C09138=1210.781,-60.471,-39.584,179.733,5.457,149.035
C09139=1210.776,-60.222,-39.597,179.735,5.458,149.035
C09140=1210.771,-59.972,-39.609,179.737,5.458,149.034
C09141=1210.766,-59.722,-39.620,179.739,5.458,149.033
C09142=1210.761,-59.473,-39.632,179.742,5.459,149.033
C09143=1210.755,-59.223,-39.644,179.744,5.458,149.032
C09144=1210.751,-58.973,-39.655,179.747,5.459,149.031
C09145=1210.745,-58.724,-39.668,179.750,5.459,149.031
C09146=1210.740,-58.474,-39.679,179.752,5.459,149.030
C09147=1210.735,-58.224,-39.691,179.754,5.459,149.029
C09148=1210.730,-57.974,-39.703,179.756,5.459,149.029
C09149=1210.724,-57.724,-39.715,179.759,5.460,149.028
C09150=1210.720,-57.475,-39.726,179.761,5.460,149.027
C09151=1210.715,-57.225,-39.738,179.763,5.460,149.027
C09152=1210.709,-56.976,-39.750,179.766,5.460,149.026
C09153=1210.704,-56.726,-39.761,179.769,5.461,149.025
C09154=1210.699,-56.476,-39.773,179.771,5.460,149.025
C09155=1210.693,-56.227,-39.786,179.773,5.461,149.024
C09156=1210.689,-55.978,-39.797,179.776,5.460,149.023
C09157=1210.683,-55.728,-39.809,179.778,5.461,149.022
C09158=1210.678,-55.478,-39.821,179.780,5.462,149.022
C09159=1210.673,-55.229,-39.833,179.782,5.461,149.021
C09160=1210.668,-54.979,-39.845,179.785,5.462,149.021
C09161=1210.663,-54.729,-39.857,179.788,5.462,149.020
C09162=1210.657,-54.479,-39.868,179.790,5.462,149.019
C09163=1210.653,-54.230,-39.880,179.793,5.462,149.018
C09164=1210.647,-53.980,-39.892,179.795,5.462,149.018
C09165=1210.642,-53.730,-39.904,179.797,5.463,149.017
C09166=1210.637,-53.481,-39.917,179.800,5.463,149.016
C09167=1210.632,-53.231,-39.928,179.802,5.463,149.016
C09168=1210.627,-52.981,-39.940,179.804,5.464,149.015
C09169=1210.622,-52.732,-39.953,179.807,5.464,149.014
C09170=1210.616,-52.482,-39.964,179.809,5.464,149.014
C09171=1210.611,-52.232,-39.976,179.812,5.464,149.013
C09172=1210.606,-51.983,-39.988,179.814,5.464,149.012
C09173=1210.601,-51.733,-40.000,179.816,5.464,149.012
C09174=1210.596,-51.484,-40.013,179.819,5.465,149.011
C09175=1210.590,-51.234,-40.025,179.821,5.464,149.010
C09176=1210.586,-50.984,-40.036,179.824,5.465,149.010
C09177=1210.581,-50.735,-40.049,179.826,5.465,149.009
C09178=1210.575,-50.485,-40.060,179.828,5.465,149.008
C09179=1210.570,-50.236,-40.073,179.831,5.466,149.008
C09180=1210.565,-49.986,-40.085,179.833,5.466,149.007
C09181=1210.559,-49.736,-40.097,179.835,5.466,149.006
C09182=1210.555,-49.487,-40.109,179.838,5.466,149.006
C09183=1210.549,-49.216,-40.122,179.841,5.467,149.005
C09184=1210.543,-48.946,-40.135,179.843,5.466,149.004
C09185=1210.538,-48.677,-40.149,179.846,5.467,149.003
C09186=1210.532,-48.406,-40.162,179.849,5.467,149.002
C09187=1210.527,-48.156,-40.174,179.851,5.468,149.002
C09188=1210.522,-47.907,-40.186,179.853,5.467,149.001
C09189=1210.516,-47.657,-40.198,179.856,5.468,149.001
C09190=1210.511,-47.408,-40.211,179.858,5.468,149.000
C09191=1210.506,-47.158,-40.223,179.860,5.468,148.999
C09192=1210.502,-46.909,-40.235,179.863,5.469,148.998
C09193=1210.497,-46.658,-40.247,179.865,5.468,148.998
C09194=1210.492,-46.409,-40.259,179.868,5.469,148.997
C09195=1210.486,-46.159,-40.271,179.870,5.469,148.996
C09196=1210.481,-45.910,-40.284,179.873,5.469,148.996
C09197=1210.476,-45.660,-40.296,179.875,5.469,148.995
C09198=1210.470,-45.410,-40.308,179.877,5.470,148.995
C09199=1210.465,-45.161,-40.321,179.879,5.470,148.994
C09200=1210.460,-44.911,-40.333,179.882,5.470,148.993
C09201=1210.455,-44.662,-40.345,179.885,5.471,148.992
C09202=1210.449,-44.412,-40.357,179.887,5.470,148.992
C09203=1210.445,-44.162,-40.370,179.890,5.471,148.991
C09204=1210.440,-43.912,-40.383,179.892,5.471,148.990
C09205=1210.434,-43.663,-40.395,179.894,5.471,148.990
C09206=1210.429,-43.413,-40.407,179.897,5.471,148.989
C09207=1210.424,-43.163,-40.419,179.900,5.472,148.988
C09208=1210.419,-42.914,-40.432,179.901,5.472,148.988
C09209=1210.413,-42.665,-40.444,179.904,5.472,148.987
C09210=1210.409,-42.414,-40.457,179.907,5.473,148.986
C09211=1210.404,-42.165,-40.469,179.909,5.473,148.986
C09212=1210.398,-41.915,-40.482,179.911,5.473,148.985
C09213=1210.393,-41.665,-40.494,179.914,5.473,148.984
C09214=1210.388,-41.416,-40.506,179.916,5.473,148.984
C09215=1210.383,-41.167,-40.519,179.919,5.474,148.983
C09216=1210.378,-40.916,-40.531,179.921,5.474,148.982
C09217=1210.373,-40.667,-40.544,179.923,5.474,148.981
C09218=1210.368,-40.418,-40.556,179.926,5.474,148.981
C09219=1210.362,-40.168,-40.568,179.928,5.475,148.980
C09220=1210.357,-39.918,-40.581,179.930,5.475,148.980
C09221=1210.352,-39.669,-40.594,179.933,5.475,148.979
C09222=1210.347,-39.419,-40.607,179.936,5.476,148.978
C09223=1210.342,-39.169,-40.618,179.938,5.475,148.977
C09224=1210.337,-38.920,-40.631,179.940,5.476,148.977
C09225=1210.332,-38.670,-40.644,179.943,5.476,148.976
C09226=1210.327,-38.421,-40.656,179.945,5.476,148.975
C09227=1210.322,-38.170,-40.668,179.948,5.476,148.975
C09228=1210.317,-37.921,-40.681,179.950,5.477,148.974
C09229=1210.312,-37.672,-40.694,179.952,5.477,148.973
C09230=1210.306,-37.422,-40.707,179.955,5.477,148.973
C09231=1210.300,-37.172,-40.719,179.957,5.478,148.972
C09232=1210.296,-36.922,-40.732,179.959,5.477,148.971
C09233=1210.291,-36.673,-40.744,179.962,5.478,148.971
C09234=1210.286,-36.424,-40.757,179.965,5.478,148.970
C09235=1210.280,-36.174,-40.770,179.967,5.479,148.969
C09236=1210.276,-35.924,-40.782,179.970,5.479,148.969
C09237=1210.270,-35.674,-40.794,179.972,5.479,148.968
C09238=1210.265,-35.425,-40.808,179.975,5.480,148.967
C09239=1210.259,-35.175,-40.820,179.977,5.479,148.966
C09240=1210.255,-34.925,-40.833,179.979,5.480,148.966
C09241=1210.250,-34.676,-40.846,179.982,5.481,148.965
C09242=1210.245,-34.427,-40.858,179.984,5.480,148.965
C09243=1210.240,-34.177,-40.871,179.987,5.481,148.964
C09244=1210.234,-33.926,-40.884,179.989,5.481,148.963
C09245=1210.229,-33.677,-40.896,179.991,5.481,148.963
C09246=1210.224,-33.428,-40.909,179.994,5.481,148.962
C09247=1210.219,-33.178,-40.922,179.997,5.482,148.961
C09248=1210.214,-32.928,-40.935,179.999,5.482,148.960
C09249=1210.209,-32.679,-40.947,-179.999,5.482,148.960
C09250=1210.203,-32.430,-40.960,-179.996,5.482,148.959
C09251=1210.199,-32.179,-40.973,-179.994,5.483,148.959
C09252=1210.193,-31.930,-40.986,-179.992,5.483,148.958
C09253=1210.188,-31.681,-40.999,-179.989,5.483,148.957
C09254=1210.182,-31.431,-41.012,-179.986,5.484,148.956
C09255=1210.178,-31.181,-41.025,-179.984,5.484,148.956
C09256=1210.173,-30.932,-41.037,-179.982,5.484,148.955
C09257=1210.168,-30.683,-41.050,-179.979,5.484,148.954
C09258=1210.163,-30.433,-41.063,-179.976,5.485,148.954
C09259=1210.157,-30.183,-41.076,-179.974,5.485,148.953
C09260=1210.152,-29.934,-41.089,-179.972,5.485,148.952
C09261=1210.148,-29.684,-41.102,-179.969,5.486,148.952
C09262=1210.142,-29.434,-41.115,-179.967,5.486,148.951
C09263=1210.137,-29.185,-41.127,-179.965,5.486,148.950
C09264=1210.132,-28.935,-41.140,-179.962,5.487,148.950
C09265=1210.127,-28.685,-41.153,-179.960,5.486,148.949
C09266=1210.121,-28.436,-41.166,-179.957,5.487,148.948
C09267=1210.117,-28.186,-41.179,-179.955,5.487,148.948
C09268=1210.112,-27.936,-41.192,-179.952,5.488,148.947
C09269=1210.106,-27.687,-41.205,-179.950,5.487,148.946
C09270=1210.101,-27.437,-41.218,-179.947,5.488,148.946
C09271=1210.096,-27.187,-41.230,-179.945,5.488,148.945
C09272=1210.091,-26.939,-41.244,-179.942,5.489,148.944
C09273=1210.086,-26.688,-41.257,-179.940,5.489,148.944
C09274=1210.081,-26.439,-41.270,-179.938,5.489,148.943
C09275=1210.076,-26.189,-41.283,-179.935,5.490,148.942
C09276=1210.070,-25.939,-41.296,-179.933,5.489,148.942
C09277=1210.065,-25.690,-41.309,-179.930,5.490,148.941
C09278=1210.060,-25.440,-41.322,-179.928,5.490,148.940
C09279=1210.055,-25.190,-41.335,-179.925,5.491,148.939
C09280=1210.051,-24.941,-41.349,-179.923,5.491,148.939
C09281=1210.045,-24.691,-41.362,-179.920,5.491,148.938
C09282=1210.040,-24.442,-41.374,-179.918,5.492,148.937
C09283=1210.035,-24.192,-41.387,-179.916,5.492,148.937
C09284=1210.029,-23.942,-41.401,-179.913,5.492,148.936
C09285=1210.025,-23.693,-41.414,-179.911,5.493,148.936
C09286=1210.019,-23.443,-41.427,-179.908,5.493,148.935
C09287=1210.014,-23.174,-41.441,-179.905,5.494,148.934
C09288=1210.008,-22.905,-41.456,-179.903,5.493,148.933
C09289=1210.003,-22.635,-41.469,-179.900,5.493,148.933
C09290=1209.998,-22.365,-41.484,-179.897,5.494,148.932
C09291=1209.993,-22.117,-41.497,-179.895,5.494,148.931
C09292=1209.987,-21.866,-41.511,-179.892,5.495,148.930
C09293=1209.982,-21.617,-41.523,-179.891,5.495,148.930
C09294=1209.977,-21.367,-41.537,-179.888,5.495,148.929
C09295=1209.972,-21.118,-41.550,-179.885,5.496,148.929
C09296=1209.966,-20.868,-41.563,-179.883,5.496,148.928
C09297=1209.962,-20.618,-41.576,-179.880,5.496,148.927
C09298=1209.956,-20.369,-41.590,-179.878,5.496,148.926
C09299=1209.952,-20.119,-41.603,-179.875,5.497,148.926
C09300=1209.946,-19.870,-41.616,-179.872,5.497,148.925
C09301=1209.942,-19.620,-41.630,-179.870,5.497,148.924
C09302=1209.937,-19.371,-41.643,-179.868,5.498,148.924
C09303=1209.931,-19.120,-41.656,-179.865,5.498,148.923
C09304=1209.926,-18.872,-41.669,-179.863,5.499,148.923
C09305=1209.921,-18.621,-41.683,-179.861,5.499,148.922
C09306=1209.915,-18.372,-41.696,-179.858,5.499,148.921
C09307=1209.911,-18.122,-41.710,-179.856,5.500,148.920
C09308=1209.905,-17.873,-41.723,-179.853,5.500,148.920
C09309=1209.901,-17.623,-41.736,-179.851,5.500,148.919
C09310=1209.895,-17.374,-41.750,-179.848,5.500,148.918
C09311=1209.891,-17.124,-41.763,-179.845,5.501,148.918
C09312=1209.885,-16.875,-41.777,-179.843,5.501,148.917
C09313=1209.881,-16.625,-41.790,-179.841,5.501,148.916
C09314=1209.875,-16.376,-41.804,-179.839,5.502,148.916
C09315=1209.871,-16.126,-41.817,-179.836,5.502,148.915
C09316=1209.865,-15.876,-41.830,-179.833,5.503,148.914
C09317=1209.860,-15.627,-41.844,-179.831,5.502,148.914
C09318=1209.855,-15.377,-41.857,-179.829,5.503,148.913
C09319=1209.850,-15.127,-41.871,-179.826,5.503,148.912
C09320=1209.844,-14.878,-41.884,-179.823,5.504,148.912
C09321=1209.840,-14.628,-41.898,-179.821,5.504,148.911
C09322=1209.834,-14.379,-41.910,-179.818,5.504,148.910
C09323=1209.829,-14.129,-41.925,-179.816,5.505,148.910
C09324=1209.824,-13.879,-41.938,-179.814,5.505,148.909
C09325=1209.819,-13.630,-41.952,-179.811,5.506,148.908
C09326=1209.814,-13.380,-41.965,-179.809,5.506,148.908
C09327=1209.809,-13.131,-41.979,-179.806,5.506,148.907
C09328=1209.804,-12.881,-41.992,-179.804,5.507,148.906
C09329=1209.798,-12.632,-42.006,-179.801,5.507,148.906
C09330=1209.794,-12.382,-42.019,-179.799,5.507,148.905
C09331=1209.789,-12.132,-42.033,-179.796,5.507,148.904
C09332=1209.783,-11.883,-42.047,-179.794,5.508,148.904
C09333=1209.779,-11.633,-42.060,-179.791,5.508,148.903
C09334=1209.773,-11.384,-42.074,-179.789,5.508,148.902
C09335=1209.768,-11.134,-42.088,-179.787,5.509,148.902
C09336=1209.763,-10.885,-42.101,-179.784,5.509,148.901
C09337=1209.758,-10.635,-42.115,-179.781,5.510,148.900
C09338=1209.753,-10.385,-42.129,-179.779,5.510,148.900
C09339=1209.748,-10.136,-42.142,-179.777,5.510,148.899
C09340=1209.743,-9.886,-42.156,-179.774,5.510,148.898
C09341=1209.738,-9.636,-42.170,-179.771,5.511,148.898
C09342=1209.733,-9.388,-42.183,-179.769,5.511,148.897
C09343=1209.728,-9.137,-42.197,-179.766,5.512,148.896
C09344=1209.722,-8.888,-42.211,-179.764,5.512,148.896
C09345=1209.717,-8.639,-42.225,-179.762,5.512,148.895
C09346=1209.713,-8.389,-42.238,-179.759,5.513,148.894
C09347=1209.707,-8.140,-42.252,-179.756,5.513,148.894
C09348=1209.702,-7.890,-42.266,-179.754,5.513,148.893
C09349=1209.697,-7.639,-42.280,-179.752,5.514,148.892
C09350=1209.692,-7.391,-42.293,-179.749,5.514,148.892
C09351=1209.687,-7.141,-42.307,-179.746,5.515,148.891
C09352=1209.682,-6.891,-42.322,-179.744,5.515,148.890
C09353=1209.677,-6.642,-42.335,-179.742,5.515,148.890
C09354=1209.672,-6.392,-42.348,-179.739,5.516,148.889
C09355=1209.667,-6.143,-42.363,-179.737,5.516,148.888
C09356=1209.662,-5.894,-42.377,-179.734,5.517,148.888
C09357=1209.657,-5.643,-42.390,-179.732,5.517,148.887
C09358=1209.652,-5.394,-42.404,-179.729,5.517,148.886
C09359=1209.647,-5.145,-42.418,-179.727,5.517,148.886
C09360=1209.642,-4.895,-42.432,-179.724,5.518,148.885
C09361=1209.637,-4.645,-42.446,-179.721,5.518,148.884
C09362=1209.631,-4.396,-42.460,-179.719,5.519,148.884
C09363=1209.626,-4.146,-42.474,-179.717,5.520,148.883
C09364=1209.622,-3.897,-42.487,-179.715,5.519,148.882
C09365=1209.616,-3.648,-42.501,-179.712,5.520,148.882
C09366=1209.611,-3.397,-42.515,-179.709,5.520,148.881
C09367=1209.606,-3.148,-42.529,-179.707,5.521,148.880
C09368=1209.601,-2.898,-42.544,-179.704,5.521,148.880
C09369=1209.596,-2.649,-42.557,-179.702,5.521,148.879
C09370=1209.591,-2.400,-42.571,-179.699,5.522,148.878
C09371=1209.586,-2.150,-42.585,-179.697,5.522,148.878
C09372=1209.581,-1.901,-42.599,-179.694,5.523,148.877
C09373=1209.576,-1.651,-42.614,-179.692,5.523,148.876
C09374=1209.571,-1.401,-42.627,-179.690,5.523,148.876
C09375=1209.566,-1.151,-42.641,-179.687,5.524,148.875
C09376=1209.560,-0.902,-42.655,-179.684,5.524,148.874
C09377=1209.555,-0.652,-42.670,-179.682,5.525,148.874
C09378=1209.550,-0.403,-42.684,-179.679,5.525,148.873
C09379=1209.546,-0.153,-42.698,-179.676,5.526,148.872
C09380=1209.540,0.096,-42.711,-179.674,5.525,148.872
C09381=1209.536,0.345,-42.726,-179.672,5.526,148.871
C09382=1209.531,0.595,-42.740,-179.670,5.527,148.870
C09383=1209.526,0.845,-42.754,-179.667,5.527,148.870
C09384=1209.520,1.094,-42.768,-179.664,5.528,148.869
C09385=1209.515,1.344,-42.782,-179.662,5.528,148.868
C09386=1209.510,1.593,-42.797,-179.660,5.528,148.868
C09387=1209.505,1.843,-42.811,-179.657,5.528,148.867
C09388=1209.500,2.093,-42.825,-179.654,5.529,148.866
C09389=1209.495,2.342,-42.839,-179.652,5.529,148.866
C09390=1209.490,2.591,-42.854,-179.649,5.530,148.865
C09391=1209.484,2.861,-42.869,-179.646,5.530,148.864
C09392=1209.479,3.130,-42.884,-179.644,5.531,148.864
C09393=1209.474,3.399,-42.899,-179.641,5.532,148.863
C09394=1209.469,3.668,-42.915,-179.638,5.532,148.862
C09395=1209.463,3.917,-42.929,-179.636,5.532,148.861
C09396=1209.458,4.167,-42.943,-179.634,5.532,148.861
C09397=1209.453,4.416,-42.957,-179.631,5.533,148.860
C09398=1209.448,4.666,-42.972,-179.629,5.534,148.860
C09399=1209.443,4.916,-42.986,-179.626,5.534,148.859
C09400=1209.438,5.165,-43.000,-179.623,5.535,148.858
C09401=1209.433,5.414,-43.014,-179.621,5.535,148.858
C09402=1209.428,5.664,-43.029,-179.619,5.535,148.857
C09403=1209.423,5.913,-43.043,-179.616,5.535,148.856
C09404=1209.417,6.163,-43.058,-179.613,5.536,148.856
C09405=1209.412,6.413,-43.073,-179.611,5.536,148.855
C09406=1209.407,6.663,-43.087,-179.609,5.537,148.854
C09407=1209.403,6.912,-43.101,-179.606,5.538,148.854
C09408=1209.397,7.161,-43.115,-179.603,5.538,148.853
C09409=1209.392,7.411,-43.130,-179.601,5.538,148.852
C09410=1209.387,7.660,-43.144,-179.599,5.538,148.852
C09411=1209.382,7.910,-43.159,-179.596,5.539,148.851
C09412=1209.377,8.160,-43.173,-179.593,5.539,148.850
C09413=1209.373,8.409,-43.187,-179.591,5.540,148.850
C09414=1209.368,8.658,-43.202,-179.588,5.541,148.849
C09415=1209.363,8.908,-43.216,-179.586,5.541,148.848
C09416=1209.357,9.157,-43.231,-179.584,5.541,148.848
C09417=1209.352,9.407,-43.245,-179.581,5.542,148.847
C09418=1209.347,9.656,-43.260,-179.578,5.542,148.846
C09419=1209.342,9.906,-43.274,-179.576,5.543,148.846
C09420=1209.337,10.156,-43.289,-179.573,5.543,148.845
C09421=1209.332,10.405,-43.303,-179.571,5.544,148.845
C09422=1209.328,10.654,-43.318,-179.568,5.544,148.844
C09423=1209.322,10.905,-43.333,-179.566,5.544,148.843
C09424=1209.317,11.154,-43.347,-179.564,5.545,148.843
C09425=1209.312,11.403,-43.362,-179.561,5.545,148.842
C09426=1209.307,11.653,-43.376,-179.558,5.546,148.841
C09427=1209.302,11.902,-43.390,-179.556,5.546,148.840
C09428=1209.296,12.152,-43.405,-179.553,5.547,148.840
C09429=1209.291,12.401,-43.420,-179.551,5.548,148.839
C09430=1209.286,12.651,-43.434,-179.548,5.548,148.839
C09431=1209.282,12.900,-43.449,-179.546,5.549,148.838
C09432=1209.277,13.150,-43.464,-179.543,5.548,148.837
C09433=1209.271,13.400,-43.479,-179.541,5.549,148.837
C09434=1209.266,13.649,-43.494,-179.538,5.549,148.836
C09435=1209.262,13.898,-43.508,-179.536,5.550,148.835
C09436=1209.257,14.148,-43.522,-179.533,5.551,148.835
C09437=1209.252,14.397,-43.537,-179.531,5.551,148.834
C09438=1209.246,14.647,-43.552,-179.528,5.552,148.833
C09439=1209.242,14.896,-43.567,-179.525,5.552,148.833
C09440=1209.237,15.146,-43.581,-179.523,5.552,148.832
C09441=1209.231,15.396,-43.597,-179.521,5.553,148.831
C09442=1209.226,15.645,-43.611,-179.518,5.553,148.831
C09443=1209.221,15.895,-43.625,-179.516,5.554,148.830
C09444=1209.217,16.144,-43.640,-179.513,5.554,148.830
C09445=1209.211,16.394,-43.655,-179.511,5.555,148.829
C09446=1209.206,16.643,-43.670,-179.508,5.556,148.828
C09447=1209.201,16.893,-43.685,-179.505,5.556,148.827
C09448=1209.196,17.142,-43.700,-179.503,5.557,148.827
C09449=1209.191,17.392,-43.714,-179.500,5.557,148.826
C09450=1209.186,17.641,-43.729,-179.498,5.557,148.825
C09451=1209.181,17.891,-43.744,-179.496,5.558,148.825
C09452=1209.176,18.140,-43.759,-179.493,5.558,148.824
C09453=1209.171,18.390,-43.774,-179.490,5.559,148.824
C09454=1209.166,18.639,-43.789,-179.488,5.559,148.823
C09455=1209.161,18.889,-43.803,-179.485,5.560,148.822
C09456=1209.156,19.138,-43.818,-179.483,5.560,148.822
C09457=1209.151,19.387,-43.834,-179.480,5.561,148.821
C09458=1209.146,19.637,-43.848,-179.478,5.562,148.820
C09459=1209.141,19.886,-43.863,-179.475,5.562,148.820
C09460=1209.135,20.136,-43.878,-179.472,5.563,148.819
C09461=1209.131,20.385,-43.893,-179.470,5.562,148.818
C09462=1209.127,20.635,-43.908,-179.468,5.563,148.818
C09463=1209.121,20.885,-43.923,-179.465,5.563,148.817
C09464=1209.116,21.134,-43.938,-179.463,5.564,148.817
C09465=1209.111,21.384,-43.953,-179.460,5.565,148.816
C09466=1209.106,21.633,-43.968,-179.458,5.565,148.815
C09467=1209.101,21.883,-43.983,-179.455,5.566,148.815
C09468=1209.096,22.133,-43.998,-179.452,5.566,148.814
C09469=1209.091,22.382,-44.013,-179.450,5.567,148.813
C09470=1209.086,22.631,-44.029,-179.447,5.567,148.812
C09471=1209.081,22.881,-44.043,-179.445,5.568,148.812
C09472=1209.075,23.130,-44.059,-179.442,5.569,148.811
C09473=1209.071,23.380,-44.074,-179.440,5.569,148.811
C09474=1209.066,23.630,-44.088,-179.438,5.569,148.810
C09475=1209.061,23.879,-44.104,-179.435,5.570,148.809
C09476=1209.056,24.128,-44.119,-179.432,5.570,148.809
C09477=1209.051,24.378,-44.134,-179.430,5.571,148.808
C09478=1209.046,24.627,-44.149,-179.427,5.572,148.807
C09479=1209.041,24.877,-44.164,-179.425,5.572,148.807
C09480=1209.036,25.126,-44.179,-179.422,5.573,148.806
C09481=1209.031,25.376,-44.195,-179.419,5.573,148.805
C09482=1209.026,25.626,-44.209,-179.417,5.574,148.805
C09483=1209.021,25.875,-44.225,-179.415,5.575,148.804
C09484=1209.016,26.124,-44.240,-179.412,5.575,148.804
C09485=1209.011,26.373,-44.256,-179.409,5.576,148.803
C09486=1209.006,26.623,-44.271,-179.407,5.576,148.802
C09487=1209.000,26.873,-44.285,-179.404,5.577,148.802
C09488=1208.996,27.122,-44.301,-179.401,5.577,148.801
C09489=1208.991,27.372,-44.316,-179.399,5.578,148.800
C09490=1208.986,27.621,-44.332,-179.397,5.578,148.800
C09491=1208.981,27.870,-44.347,-179.395,5.578,148.799
C09492=1208.976,28.120,-44.363,-179.392,5.579,148.798
C09493=1208.971,28.369,-44.377,-179.389,5.579,148.798
C09494=1208.966,28.619,-44.393,-179.387,5.580,148.797
C09495=1208.961,28.888,-44.409,-179.384,5.580,148.796
C09496=1208.955,29.157,-44.426,-179.381,5.582,148.796
C09497=1208.950,29.425,-44.443,-179.378,5.582,148.795
C09498=1208.944,29.694,-44.458,-179.375,5.583,148.794
C09499=1208.939,29.943,-44.474,-179.373,5.583,148.794
C09500=1208.934,30.193,-44.489,-179.371,5.584,148.793
C09501=1208.930,30.443,-44.505,-179.368,5.585,148.793
C09502=1208.924,30.692,-44.520,-179.365,5.585,148.792
C09503=1208.920,30.941,-44.535,-179.363,5.586,148.791
C09504=1208.914,31.191,-44.551,-179.361,5.586,148.791
C09505=1208.909,31.440,-44.567,-179.358,5.586,148.790
C09506=1208.905,31.690,-44.582,-179.356,5.587,148.789
C09507=1208.899,31.939,-44.597,-179.353,5.587,148.789
C09508=1208.894,32.189,-44.613,-179.351,5.588,148.788
C09509=1208.889,32.438,-44.628,-179.348,5.589,148.787
C09510=1208.885,32.688,-44.644,-179.345,5.589,148.787
C09511=1208.879,32.937,-44.660,-179.343,5.590,148.786
C09512=1208.874,33.186,-44.675,-179.341,5.590,148.786
C09513=1208.869,33.436,-44.690,-179.338,5.591,148.785
C09514=1208.864,33.686,-44.706,-179.335,5.592,148.784
C09515=1208.860,33.935,-44.721,-179.333,5.592,148.784
C09516=1208.854,34.184,-44.737,-179.330,5.593,148.783
C09517=1208.849,34.434,-44.753,-179.328,5.594,148.782
C09518=1208.845,34.683,-44.768,-179.325,5.594,148.782
C09519=1208.839,34.933,-44.783,-179.323,5.595,148.781
C09520=1208.834,35.182,-44.800,-179.320,5.595,148.780
C09521=1208.830,35.432,-44.816,-179.317,5.596,148.780
C09522=1208.825,35.681,-44.831,-179.315,5.597,148.779
C09523=1208.820,35.930,-44.846,-179.312,5.597,148.779
C09524=1208.815,36.180,-44.862,-179.310,5.598,148.778
C09525=1208.809,36.430,-44.878,-179.307,5.598,148.777
C09526=1208.805,36.679,-44.893,-179.305,5.599,148.777
C09527=1208.800,36.929,-44.909,-179.302,5.600,148.776
C09528=1208.795,37.178,-44.925,-179.300,5.600,148.775
C09529=1208.789,37.427,-44.940,-179.297,5.601,148.775
C09530=1208.784,37.676,-44.956,-179.294,5.601,148.774
C09531=1208.780,37.926,-44.971,-179.292,5.602,148.773
C09532=1208.775,38.176,-44.987,-179.289,5.602,148.773
C09533=1208.769,38.425,-45.003,-179.287,5.603,148.772
C09534=1208.765,38.675,-45.019,-179.284,5.604,148.772
C09535=1208.759,38.924,-45.035,-179.282,5.604,148.771
C09536=1208.755,39.173,-45.050,-179.279,5.605,148.770
C09537=1208.750,39.423,-45.066,-179.276,5.605,148.770
C09538=1208.745,39.672,-45.082,-179.274,5.606,148.769
C09539=1208.740,39.922,-45.098,-179.272,5.607,148.769
C09540=1208.735,40.171,-45.114,-179.269,5.607,148.768
C09541=1208.729,40.421,-45.129,-179.266,5.608,148.767
C09542=1208.726,40.670,-45.145,-179.264,5.608,148.766
C09543=1208.720,40.919,-45.161,-179.262,5.609,148.766
C09544=1208.715,41.169,-45.176,-179.259,5.610,148.765
C09545=1208.710,41.419,-45.192,-179.256,5.610,148.765
C09546=1208.705,41.668,-45.209,-179.254,5.611,148.764
C09547=1208.700,41.918,-45.225,-179.251,5.611,148.763
C09548=1208.695,42.167,-45.240,-179.249,5.612,148.763
C09549=1208.690,42.416,-45.257,-179.246,5.613,148.762
C09550=1208.685,42.666,-45.273,-179.244,5.613,148.762
C09551=1208.680,42.915,-45.288,-179.241,5.614,148.761
C09552=1208.676,43.165,-45.304,-179.239,5.615,148.760
C09553=1208.670,43.414,-45.320,-179.236,5.615,148.760
C09554=1208.665,43.663,-45.336,-179.234,5.616,148.759
C09555=1208.661,43.913,-45.352,-179.231,5.616,148.758
C09556=1208.655,44.162,-45.368,-179.228,5.617,148.758
C09557=1208.651,44.412,-45.384,-179.226,5.618,148.757
C09558=1208.645,44.661,-45.400,-179.223,5.618,148.757
C09559=1208.641,44.911,-45.417,-179.221,5.619,148.756
C09560=1208.635,45.160,-45.432,-179.218,5.619,148.755
C09561=1208.630,45.410,-45.448,-179.215,5.621,148.755
C09562=1208.626,45.659,-45.464,-179.213,5.622,148.754
C09563=1208.620,45.908,-45.480,-179.210,5.622,148.754
C09564=1208.616,46.158,-45.497,-179.208,5.623,148.753
C09565=1208.610,46.407,-45.512,-179.205,5.623,148.752
C09566=1208.606,46.657,-45.529,-179.203,5.624,148.752
C09567=1208.600,46.906,-45.545,-179.200,5.625,148.751
C09568=1208.596,47.156,-45.561,-179.197,5.625,148.750
C09569=1208.591,47.405,-45.577,-179.195,5.626,148.750
C09570=1208.586,47.655,-45.593,-179.192,5.626,148.749
C09571=1208.581,47.904,-45.609,-179.190,5.627,148.749
C09572=1208.576,48.153,-45.626,-179.187,5.628,148.748
C09573=1208.571,48.403,-45.641,-179.185,5.628,148.747
C09574=1208.566,48.652,-45.658,-179.182,5.629,148.747
C09575=1208.561,48.902,-45.674,-179.180,5.630,148.746
C09576=1208.556,49.151,-45.690,-179.177,5.630,148.745
C09577=1208.551,49.400,-45.707,-179.175,5.631,148.745
C09578=1208.547,49.650,-45.722,-179.172,5.631,148.744
C09579=1208.542,49.899,-45.739,-179.170,5.632,148.744
C09580=1208.537,50.149,-45.755,-179.167,5.633,148.743
C09581=1208.532,50.398,-45.771,-179.165,5.633,148.742
C09582=1208.527,50.647,-45.788,-179.161,5.635,148.742
C09583=1208.521,50.897,-45.804,-179.159,5.635,148.741
C09584=1208.517,51.146,-45.821,-179.157,5.636,148.741
C09585=1208.511,51.396,-45.836,-179.154,5.637,148.740
C09586=1208.507,51.645,-45.853,-179.151,5.637,148.739
C09587=1208.502,51.894,-45.869,-179.149,5.638,148.739
C09588=1208.497,52.144,-45.885,-179.147,5.639,148.738
C09589=1208.492,52.394,-45.902,-179.144,5.639,148.737
C09590=1208.487,52.642,-45.918,-179.141,5.640,148.737
C09591=1208.482,52.893,-45.935,-179.139,5.640,148.736
C09592=1208.477,53.142,-45.951,-179.137,5.641,148.736
C09593=1208.472,53.391,-45.968,-179.134,5.642,148.735
C09594=1208.467,53.640,-45.984,-179.131,5.642,148.734
C09595=1208.462,53.890,-46.000,-179.129,5.643,148.734
C09596=1208.458,54.140,-46.016,-179.126,5.645,148.733
C09597=1208.452,54.389,-46.033,-179.123,5.645,148.733
C09598=1208.448,54.638,-46.050,-179.121,5.646,148.732
C09599=1208.442,54.907,-46.067,-179.118,5.646,148.731
C09600=1208.437,55.175,-46.085,-179.115,5.647,148.731
C09601=1208.431,55.444,-46.103,-179.113,5.648,148.730
C09602=1208.426,55.712,-46.121,-179.110,5.649,148.729
C09603=1208.421,55.961,-46.137,-179.107,5.650,148.729
C09604=1208.417,56.211,-46.154,-179.105,5.650,148.728
C09605=1208.411,56.460,-46.170,-179.102,5.651,148.727
C09606=1208.406,56.710,-46.187,-179.099,5.651,148.727
C09607=1208.401,56.959,-46.203,-179.097,5.652,148.726
C09608=1208.397,57.208,-46.220,-179.095,5.653,148.726
C09609=1208.391,57.458,-46.237,-179.092,5.653,148.725
C09610=1208.386,57.707,-46.253,-179.089,5.654,148.724
C09611=1208.382,57.957,-46.269,-179.087,5.656,148.724
C09612=1208.377,58.206,-46.286,-179.084,5.656,148.723
C09613=1208.371,58.456,-46.303,-179.081,5.657,148.723
C09614=1208.367,58.705,-46.319,-179.079,5.657,148.722
C09615=1208.362,58.954,-46.336,-179.077,5.658,148.722
C09616=1208.357,59.204,-46.353,-179.074,5.659,148.721
C09617=1208.352,59.453,-46.370,-179.071,5.659,148.720
C09618=1208.348,59.703,-46.386,-179.069,5.660,148.720
C09619=1208.342,59.951,-46.403,-179.067,5.661,148.719
C09620=1208.337,60.201,-46.420,-179.064,5.661,148.718
C09621=1208.333,60.451,-46.437,-179.061,5.663,148.718
C09622=1208.328,60.699,-46.453,-179.059,5.664,148.717
C09623=1208.322,60.949,-46.470,-179.056,5.664,148.717
C09624=1208.318,61.199,-46.487,-179.053,5.665,148.716
C09625=1208.312,61.448,-46.504,-179.051,5.665,148.715
C09626=1208.308,61.697,-46.520,-179.049,5.666,148.715
C09627=1208.303,61.947,-46.537,-179.046,5.667,148.714
C09628=1208.298,62.197,-46.554,-179.043,5.667,148.714
C09629=1208.293,62.445,-46.571,-179.040,5.669,148.713
C09630=1208.288,62.695,-46.587,-179.038,5.670,148.712
C09631=1208.283,62.945,-46.605,-179.035,5.670,148.712
C09632=1208.278,63.193,-46.621,-179.033,5.671,148.711
C09633=1208.273,63.443,-46.638,-179.031,5.672,148.711
C09634=1208.268,63.693,-46.655,-179.028,5.672,148.710
C09635=1208.264,63.942,-46.671,-179.025,5.673,148.709
C09636=1208.258,64.191,-46.688,-179.023,5.673,148.709
C09637=1208.254,64.441,-46.705,-179.020,5.675,148.708
C09638=1208.248,64.691,-46.722,-179.017,5.676,148.708
C09639=1208.244,64.940,-46.739,-179.015,5.676,148.707
C09640=1208.238,65.189,-46.756,-179.013,5.677,148.707
C09641=1208.234,65.438,-46.773,-179.010,5.678,148.706
C09642=1208.229,65.687,-46.790,-179.007,5.678,148.705
C09643=1208.224,65.937,-46.807,-179.005,5.679,148.705
C09644=1208.219,66.186,-46.823,-179.002,5.681,148.704
C09645=1208.214,66.436,-46.841,-178.999,5.681,148.703
C09646=1208.209,66.685,-46.857,-178.997,5.682,148.703
C09647=1208.205,66.934,-46.875,-178.995,5.683,148.702
C09648=1208.200,67.184,-46.892,-178.992,5.683,148.702
C09649=1208.194,67.433,-46.909,-178.989,5.684,148.701
C09650=1208.190,67.683,-46.926,-178.987,5.684,148.700
C09651=1208.185,67.932,-46.943,-178.984,5.686,148.700
C09652=1208.180,68.181,-46.960,-178.981,5.687,148.699
C09653=1208.175,68.431,-46.978,-178.979,5.687,148.699
C09654=1208.170,68.680,-46.994,-178.977,5.688,148.698
C09655=1208.165,68.930,-47.011,-178.974,5.689,148.698
C09656=1208.161,69.178,-47.028,-178.971,5.689,148.697
C09657=1208.155,69.428,-47.046,-178.969,5.691,148.696
C09658=1208.150,69.678,-47.063,-178.966,5.691,148.696
C09659=1208.146,69.927,-47.080,-178.963,5.692,148.695
C09660=1208.140,70.176,-47.097,-178.961,5.693,148.694
C09661=1208.136,70.425,-47.114,-178.959,5.693,148.694
C09662=1208.131,70.675,-47.131,-178.956,5.694,148.693
C09663=1208.126,70.924,-47.149,-178.953,5.695,148.693
C09664=1208.121,71.174,-47.166,-178.951,5.696,148.692
C09665=1208.116,71.424,-47.183,-178.948,5.697,148.692
C09666=1208.112,71.673,-47.201,-178.945,5.697,148.691
C09667=1208.106,71.922,-47.217,-178.943,5.698,148.691
C09668=1208.101,72.171,-47.235,-178.941,5.699,148.690
C09669=1208.097,72.420,-47.252,-178.937,5.700,148.689
C09670=1208.091,72.670,-47.269,-178.935,5.701,148.689
C09671=1208.087,72.919,-47.287,-178.933,5.702,148.688
C09672=1208.082,73.169,-47.304,-178.930,5.702,148.687
C09673=1208.077,73.418,-47.322,-178.928,5.703,148.687
C09674=1208.073,73.667,-47.339,-178.925,5.704,148.686
C09675=1208.067,73.917,-47.356,-178.922,5.705,148.686
C09676=1208.062,74.166,-47.374,-178.920,5.706,148.685
C09677=1208.057,74.415,-47.390,-178.917,5.707,148.685
C09678=1208.052,74.664,-47.408,-178.915,5.707,148.684
C09679=1208.047,74.914,-47.425,-178.912,5.708,148.684
C09680=1208.043,75.163,-47.443,-178.909,5.710,148.683
C09681=1208.038,75.413,-47.460,-178.907,5.710,148.682
C09682=1208.033,75.662,-47.478,-178.904,5.711,148.682
C09683=1208.028,75.912,-47.495,-178.902,5.712,148.681
C09684=1208.024,76.161,-47.513,-178.899,5.712,148.681
C09685=1208.018,76.410,-47.530,-178.896,5.714,148.680
C09686=1208.013,76.660,-47.548,-178.894,5.715,148.679
C09687=1208.009,76.909,-47.565,-178.891,5.715,148.679
C09688=1208.004,77.158,-47.583,-178.889,5.716,148.678
C09689=1207.999,77.408,-47.600,-178.886,5.717,148.678
C09690=1207.994,77.657,-47.618,-178.883,5.718,148.677
C09691=1207.989,77.905,-47.635,-178.881,5.719,148.677
C09692=1207.984,78.155,-47.652,-178.879,5.719,148.676
C09693=1207.979,78.404,-47.670,-178.876,5.720,148.675
C09694=1207.974,78.654,-47.687,-178.874,5.721,148.675
C09695=1207.969,78.903,-47.705,-178.871,5.722,148.674
C09696=1207.965,79.152,-47.723,-178.868,5.723,148.674
C09697=1207.959,79.402,-47.740,-178.866,5.724,148.673
C09698=1207.955,79.651,-47.758,-178.863,5.724,148.672
C09699=1207.950,79.900,-47.776,-178.861,5.725,148.672
C09700=1207.944,80.150,-47.793,-178.858,5.727,148.671
C09701=1207.940,80.399,-47.811,-178.855,5.727,148.671
C09702=1207.935,80.648,-47.829,-178.853,5.728,148.670
C09703=1207.930,80.917,-47.847,-178.849,5.729,148.669
C09704=1207.925,81.185,-47.867,-178.847,5.730,148.669
C09705=1207.919,81.454,-47.885,-178.845,5.731,148.668
C09706=1207.914,81.722,-47.905,-178.841,5.732,148.668
C09707=1207.909,81.972,-47.923,-178.839,5.733,148.667
C09708=1207.904,82.221,-47.940,-178.837,5.734,148.667
C09709=1207.899,82.471,-47.958,-178.834,5.734,148.666
C09710=1207.894,82.720,-47.976,-178.831,5.736,148.665
C09711=1207.890,82.969,-47.993,-178.829,5.737,148.665
C09712=1207.885,83.218,-48.011,-178.826,5.737,148.664
C09713=1207.880,83.468,-48.029,-178.823,5.738,148.664
C09714=1207.875,83.717,-48.047,-178.821,5.739,148.663
C09715=1207.870,83.966,-48.065,-178.818,5.740,148.663
C09716=1207.865,84.215,-48.083,-178.816,5.741,148.662
C09717=1207.860,84.465,-48.100,-178.813,5.741,148.661
C09718=1207.855,84.714,-48.118,-178.810,5.743,148.661
C09719=1207.850,84.963,-48.136,-178.808,5.744,148.660
C09720=1207.846,85.213,-48.154,-178.805,5.744,148.660
C09721=1207.841,85.462,-48.172,-178.803,5.745,148.659
C09722=1207.836,85.712,-48.190,-178.800,5.747,148.659
C09723=1207.831,85.961,-48.208,-178.797,5.747,148.658
C09724=1207.826,86.210,-48.225,-178.795,5.748,148.658
C09725=1207.821,86.460,-48.243,-178.793,5.749,148.657
C09726=1207.816,86.709,-48.261,-178.789,5.750,148.656
C09727=1207.811,86.958,-48.279,-178.787,5.751,148.656
C09728=1207.806,87.207,-48.297,-178.785,5.752,148.655
C09729=1207.802,87.456,-48.315,-178.782,5.752,148.655
C09730=1207.797,87.706,-48.334,-178.779,5.754,148.654
C09731=1207.792,87.955,-48.352,-178.777,5.755,148.653
C09732=1207.787,88.205,-48.370,-178.775,5.755,148.653
C09733=1207.782,88.454,-48.388,-178.772,5.756,148.652
C09734=1207.778,88.703,-48.406,-178.769,5.757,148.652
C09735=1207.773,88.952,-48.423,-178.767,5.758,148.651
C09736=1207.768,89.201,-48.441,-178.764,5.759,148.651
C09737=1207.763,89.451,-48.460,-178.761,5.761,148.650
C09738=1207.759,89.700,-48.478,-178.759,5.761,148.650
C09739=1207.754,89.950,-48.496,-178.756,5.762,148.649
C09740=1207.749,90.199,-48.514,-178.754,5.763,148.649
C09741=1207.744,90.448,-48.532,-178.751,5.764,148.648
C09742=1207.739,90.697,-48.550,-178.749,5.765,148.647
C09743=1207.735,90.947,-48.568,-178.746,5.766,148.647
C09744=1207.730,91.196,-48.586,-178.743,5.766,148.646
C09745=1207.724,91.446,-48.605,-178.741,5.768,148.646
C09746=1207.719,91.695,-48.623,-178.738,5.769,148.645
C09747=1207.714,91.944,-48.641,-178.736,5.770,148.645
C09748=1207.709,92.193,-48.659,-178.733,5.771,148.644
C09749=1207.705,92.443,-48.677,-178.730,5.772,148.643
C09750=1207.700,92.692,-48.696,-178.728,5.772,148.643
C09751=1207.695,92.941,-48.714,-178.725,5.773,148.642
C09752=1207.691,93.190,-48.732,-178.723,5.775,148.642
C09753=1207.685,93.440,-48.751,-178.720,5.775,148.641
C09754=1207.681,93.689,-48.768,-178.717,5.776,148.641
C09755=1207.676,93.938,-48.786,-178.715,5.778,148.640
C09756=1207.671,94.188,-48.804,-178.712,5.778,148.640
C09757=1207.666,94.436,-48.823,-178.710,5.779,148.639
C09758=1207.662,94.686,-48.841,-178.707,5.781,148.638
C09759=1207.656,94.936,-48.860,-178.704,5.781,148.638
C09760=1207.651,95.185,-48.878,-178.702,5.782,148.637
C09761=1207.646,95.434,-48.896,-178.699,5.783,148.637
C09762=1207.642,95.683,-48.915,-178.697,5.784,148.636
C09763=1207.637,95.933,-48.934,-178.694,5.785,148.636
C09764=1207.632,96.182,-48.952,-178.692,5.786,148.635
C09765=1207.627,96.431,-48.970,-178.689,5.787,148.635
C09766=1207.623,96.680,-48.989,-178.686,5.788,148.634
C09767=1207.618,96.929,-49.007,-178.684,5.789,148.634
C09768=1207.612,97.179,-49.025,-178.681,5.790,148.633
C09769=1207.608,97.428,-49.044,-178.679,5.791,148.633
C09770=1207.603,97.677,-49.062,-178.676,5.792,148.632
C09771=1207.598,97.927,-49.081,-178.673,5.794,148.631
C09772=1207.593,98.175,-49.100,-178.671,5.794,148.631
C09773=1207.589,98.425,-49.118,-178.668,5.795,148.630
C09774=1207.584,98.674,-49.136,-178.665,5.797,148.630
C09775=1207.579,98.923,-49.155,-178.663,5.797,148.629
C09776=1207.574,99.173,-49.174,-178.661,5.798,148.629
C09777=1207.569,99.422,-49.191,-178.658,5.799,148.628
C09778=1207.564,99.671,-49.211,-178.655,5.800,148.628
C09779=1207.560,99.921,-49.229,-178.653,5.801,148.627
C09780=1207.555,100.170,-49.247,-178.650,5.803,148.627
C09781=1207.549,100.419,-49.266,-178.647,5.803,148.626
C09782=1207.545,100.669,-49.285,-178.645,5.804,148.625
C09783=1207.541,100.918,-49.303,-178.642,5.806,148.625
C09784=1207.535,101.167,-49.322,-178.640,5.806,148.624
C09785=1207.531,101.416,-49.341,-178.637,5.807,148.624
C09786=1207.526,101.665,-49.359,-178.634,5.809,148.623
C09787=1207.520,101.915,-49.378,-178.632,5.810,148.623
C09788=1207.516,102.164,-49.397,-178.629,5.810,148.622
C09789=1207.511,102.414,-49.415,-178.627,5.812,148.622
C09790=1207.506,102.662,-49.434,-178.624,5.812,148.621
C09791=1207.502,102.912,-49.452,-178.622,5.813,148.620
C09792=1207.496,103.161,-49.472,-178.619,5.815,148.620
C09793=1207.492,103.411,-49.490,-178.616,5.815,148.619
C09794=1207.487,103.660,-49.509,-178.614,5.816,148.619
C09795=1207.482,103.908,-49.528,-178.611,5.818,148.618
C09796=1207.478,104.158,-49.546,-178.609,5.819,148.618
C09797=1207.472,104.407,-49.566,-178.606,5.819,148.617
C09798=1207.468,104.657,-49.584,-178.603,5.821,148.617
C09799=1207.463,104.906,-49.603,-178.601,5.822,148.616
C09800=1207.458,105.155,-49.621,-178.598,5.823,148.616
C09801=1207.453,105.405,-49.641,-178.596,5.824,148.615
C09802=1207.449,105.653,-49.660,-178.593,5.825,148.615
C09803=1207.444,105.903,-49.678,-178.590,5.826,148.614
C09804=1207.439,106.152,-49.697,-178.588,5.827,148.614
C09805=1207.433,106.401,-49.716,-178.585,5.828,148.613
C09806=1207.429,106.651,-49.735,-178.582,5.829,148.612
C09807=1207.424,106.919,-49.756,-178.580,5.830,148.612
C09808=1207.419,107.188,-49.776,-178.577,5.832,148.611
C09809=1207.414,107.455,-49.796,-178.574,5.832,148.611
C09810=1207.409,107.725,-49.816,-178.572,5.834,148.610
C09811=1207.403,107.974,-49.836,-178.569,5.835,148.610
C09812=1207.399,108.222,-49.854,-178.566,5.836,148.609
C09813=1207.394,108.472,-49.873,-178.564,5.837,148.609
C09814=1207.389,108.721,-49.892,-178.562,5.838,148.608
C09815=1207.384,108.970,-49.912,-178.558,5.839,148.608
C09816=1207.380,109.219,-49.930,-178.556,5.840,148.607
C09817=1207.375,109.469,-49.949,-178.553,5.842,148.607
C09818=1207.370,109.718,-49.968,-178.551,5.843,148.606
C09819=1207.365,109.967,-49.988,-178.548,5.843,148.606
C09820=1207.360,110.216,-50.007,-178.546,5.845,148.605
C09821=1207.356,110.466,-50.025,-178.543,5.846,148.604
C09822=1207.350,110.715,-50.045,-178.540,5.847,148.604
C09823=1207.346,110.964,-50.064,-178.538,5.848,148.603
C09824=1207.341,111.213,-50.083,-178.536,5.849,148.603
C09825=1207.336,111.463,-50.103,-178.532,5.850,148.602
C09826=1207.331,111.711,-50.121,-178.530,5.851,148.602
C09827=1207.326,111.961,-50.140,-178.527,5.853,148.601
C09828=1207.321,112.210,-50.160,-178.525,5.854,148.601
C09829=1207.317,112.459,-50.179,-178.522,5.854,148.600
C09830=1207.312,112.709,-50.198,-178.520,5.856,148.600
C09831=1207.307,112.958,-50.218,-178.517,5.857,148.599
C09832=1207.303,113.207,-50.237,-178.514,5.858,148.599
C09833=1207.298,113.456,-50.256,-178.512,5.859,148.598
C09834=1207.293,113.706,-50.276,-178.510,5.860,148.598
C09835=1207.288,113.955,-50.294,-178.507,5.861,148.597
C09836=1207.283,114.204,-50.313,-178.504,5.862,148.597
C09837=1207.278,114.453,-50.332,-178.501,5.864,148.596
C09838=1207.274,114.702,-50.352,-178.499,5.865,148.596
C09839=1207.269,114.952,-50.371,-178.496,5.866,148.595
C09840=1207.264,115.201,-50.390,-178.494,5.867,148.595
C09841=1207.259,115.451,-50.410,-178.491,5.868,148.594
C09842=1207.254,115.699,-50.429,-178.488,5.869,148.594
C09843=1207.250,115.949,-50.448,-178.486,5.870,148.593
C09844=1207.244,116.197,-50.468,-178.483,5.872,148.593
C09845=1207.240,116.447,-50.487,-178.481,5.872,148.592
C09846=1207.236,116.696,-50.506,-178.478,5.874,148.592
C09847=1207.230,116.945,-50.526,-178.475,5.875,148.591
C09848=1207.226,117.195,-50.545,-178.473,5.876,148.591
C09849=1207.220,117.444,-50.565,-178.470,5.877,148.590
C09850=1207.216,117.693,-50.584,-178.468,5.878,148.589
C09851=1207.211,117.942,-50.603,-178.465,5.880,148.589
C09852=1207.206,118.191,-50.623,-178.463,5.880,148.588
C09853=1207.202,118.440,-50.643,-178.460,5.882,148.588
C09854=1207.197,118.690,-50.663,-178.457,5.883,148.587
C09855=1207.192,118.939,-50.682,-178.455,5.884,148.587
C09856=1207.188,119.188,-50.701,-178.452,5.885,148.586
C09857=1207.183,119.438,-50.721,-178.450,5.886,148.586
C09858=1207.177,119.686,-50.740,-178.447,5.887,148.585
C09859=1207.173,119.936,-50.760,-178.445,5.888,148.585
C09860=1207.168,120.185,-50.780,-178.441,5.890,148.584
C09861=1207.163,120.434,-50.799,-178.439,5.891,148.584
C09862=1207.159,120.683,-50.818,-178.436,5.892,148.583
C09863=1207.154,120.933,-50.838,-178.434,5.893,148.583
C09864=1207.149,121.181,-50.857,-178.431,5.895,148.582
C09865=1207.144,121.430,-50.878,-178.429,5.896,148.582
C09866=1207.140,121.680,-50.897,-178.426,5.897,148.581
C09867=1207.134,121.929,-50.917,-178.423,5.898,148.581
C09868=1207.130,122.178,-50.936,-178.421,5.899,148.580
C09869=1207.125,122.428,-50.956,-178.418,5.900,148.580
C09870=1207.120,122.676,-50.976,-178.416,5.901,148.579
C09871=1207.115,122.926,-50.996,-178.413,5.903,148.579
C09872=1207.110,123.175,-51.015,-178.411,5.904,148.578
C09873=1207.107,123.424,-51.035,-178.408,5.905,148.578
C09874=1207.101,123.673,-51.054,-178.405,5.906,148.577
C09875=1207.097,123.922,-51.074,-178.403,5.908,148.577
C09876=1207.092,124.172,-51.094,-178.400,5.908,148.576
C09877=1207.087,124.420,-51.114,-178.397,5.910,148.576
C09878=1207.082,124.670,-51.133,-178.395,5.911,148.575
C09879=1207.077,124.919,-51.153,-178.392,5.913,148.575
C09880=1207.073,125.168,-51.173,-178.390,5.913,148.574
C09881=1207.067,125.417,-51.193,-178.387,5.915,148.574
C09882=1207.063,125.666,-51.213,-178.385,5.916,148.573
C09883=1207.058,125.916,-51.233,-178.381,5.917,148.573
C09884=1207.054,126.165,-51.252,-178.379,5.918,148.572
C09885=1207.049,126.414,-51.273,-178.377,5.920,148.572
C09886=1207.044,126.663,-51.292,-178.374,5.921,148.571
C09887=1207.039,126.912,-51.312,-178.371,5.922,148.571
C09888=1207.035,127.162,-51.332,-178.369,5.923,148.570
C09889=1207.030,127.411,-51.352,-178.366,5.925,148.570
C09890=1207.025,127.659,-51.372,-178.363,5.925,148.569
C09891=1207.020,127.909,-51.391,-178.361,5.927,148.569
C09892=1207.015,128.158,-51.412,-178.359,5.928,148.569
C09893=1207.010,128.408,-51.432,-178.355,5.930,148.568
C09894=1207.006,128.657,-51.452,-178.353,5.931,148.568
C09895=1207.001,128.906,-51.472,-178.350,5.932,148.567
C09896=1206.996,129.155,-51.492,-178.348,5.933,148.566
C09897=1206.991,129.404,-51.512,-178.345,5.935,148.566
C09898=1206.987,129.653,-51.532,-178.343,5.935,148.565
C09899=1206.982,129.903,-51.552,-178.340,5.937,148.565
C09900=1206.978,130.152,-51.572,-178.337,5.938,148.564
C09901=1206.973,130.400,-51.592,-178.335,5.939,148.564
C09902=1206.967,130.650,-51.612,-178.333,5.940,148.564
C09903=1206.963,130.899,-51.633,-178.330,5.942,148.563
C09904=1206.958,131.148,-51.652,-178.327,5.943,148.563
C09905=1206.953,131.397,-51.673,-178.325,5.945,148.562
C09906=1206.949,131.646,-51.693,-178.322,5.945,148.562
C09907=1206.944,131.896,-51.713,-178.319,5.947,148.561
C09908=1206.938,132.144,-51.733,-178.317,5.948,148.561
C09909=1206.934,132.394,-51.753,-178.314,5.949,148.560
C09910=1206.929,132.643,-51.773,-178.312,5.950,148.560
C09911=1206.924,132.912,-51.795,-178.309,5.952,148.559
C09912=1206.919,133.180,-51.817,-178.306,5.953,148.559
C09913=1206.914,133.449,-51.839,-178.303,5.955,148.558
C09914=1206.909,133.718,-51.861,-178.300,5.956,148.558
C09915=1206.904,133.967,-51.882,-178.298,5.957,148.557
C09916=1206.899,134.216,-51.901,-178.296,5.958,148.557
C09917=1206.894,134.465,-51.921,-178.292,5.960,148.556
C09918=1206.890,134.714,-51.942,-178.290,5.962,148.556
C09919=1206.885,134.963,-51.961,-178.287,5.962,148.555
C09920=1206.880,135.212,-51.982,-178.284,5.964,148.555
C09921=1206.876,135.461,-52.003,-178.282,5.965,148.554
C09922=1206.871,135.710,-52.023,-178.279,5.966,148.554
C09923=1206.866,135.960,-52.044,-178.277,5.967,148.553
C09924=1206.861,136.209,-52.064,-178.274,5.969,148.553
C09925=1206.857,136.458,-52.084,-178.272,5.970,148.552
C09926=1206.852,136.707,-52.104,-178.269,5.971,148.552
C09927=1206.847,136.956,-52.125,-178.267,5.972,148.552
C09928=1206.843,137.205,-52.146,-178.264,5.974,148.551
C09929=1206.838,137.455,-52.165,-178.261,5.976,148.551
C09930=1206.833,137.704,-52.186,-178.259,5.977,148.550
C09931=1206.828,137.953,-52.207,-178.256,5.978,148.550
C09932=1206.823,138.201,-52.227,-178.254,5.979,148.549
C09933=1206.818,138.450,-52.248,-178.251,5.980,148.549
C09934=1206.814,138.699,-52.268,-178.248,5.981,148.548
C09935=1206.809,138.948,-52.289,-178.246,5.983,148.548
C09936=1206.804,139.198,-52.309,-178.243,5.985,148.547
C09937=1206.799,139.447,-52.329,-178.240,5.986,148.547
C09938=1206.794,139.696,-52.350,-178.238,5.987,148.546
C09939=1206.790,139.945,-52.370,-178.235,5.988,148.546
C09940=1206.785,140.194,-52.391,-178.233,5.990,148.545
C09941=1206.780,140.444,-52.412,-178.230,5.991,148.545
C09942=1206.776,140.693,-52.432,-178.227,5.992,148.544
C09943=1206.771,140.942,-52.453,-178.225,5.994,148.544
C09944=1206.766,141.191,-52.474,-178.222,5.995,148.544
C09945=1206.762,141.440,-52.494,-178.219,5.996,148.543
C09946=1206.757,141.690,-52.515,-178.217,5.997,148.543
C09947=1206.753,141.939,-52.536,-178.215,5.999,148.542
C09948=1206.748,142.188,-52.557,-178.211,6.001,148.542
C09949=1206.743,142.437,-52.577,-178.209,6.002,148.541
C09950=1206.738,142.686,-52.598,-178.207,6.003,148.541
C09951=1206.733,142.935,-52.618,-178.204,6.004,148.540
C09952=1206.729,143.184,-52.640,-178.201,6.006,148.540
C09953=1206.724,143.433,-52.660,-178.199,6.008,148.539
C09954=1206.719,143.682,-52.681,-178.196,6.009,148.539
C09955=1206.715,143.931,-52.702,-178.193,6.010,148.538
C09956=1206.709,144.180,-52.723,-178.191,6.011,148.538
C09957=1206.705,144.429,-52.743,-178.189,6.013,148.538
C09958=1206.700,144.678,-52.764,-178.185,6.014,148.537
C09959=1206.695,144.927,-52.784,-178.183,6.015,148.537
C09960=1206.691,145.177,-52.806,-178.181,6.017,148.536
C09961=1206.687,145.426,-52.827,-178.178,6.018,148.536
C09962=1206.681,145.675,-52.848,-178.175,6.019,148.535
C09963=1206.677,145.924,-52.868,-178.173,6.021,148.535
C09964=1206.672,146.173,-52.889,-178.170,6.022,148.534
C09965=1206.667,146.422,-52.909,-178.167,6.024,148.534
C09966=1206.663,146.671,-52.931,-178.165,6.024,148.533
C09967=1206.658,146.920,-52.952,-178.163,6.026,148.533
C09968=1206.653,147.169,-52.972,-178.159,6.028,148.532
C09969=1206.648,147.419,-52.994,-178.157,6.029,148.532
C09970=1206.644,147.668,-53.014,-178.155,6.030,148.532
C09971=1206.639,147.916,-53.036,-178.151,6.032,148.531
C09972=1206.635,148.165,-53.056,-178.149,6.033,148.531
C09973=1206.629,148.415,-53.077,-178.147,6.035,148.530
C09974=1206.625,148.663,-53.099,-178.145,6.036,148.530
C09975=1206.620,148.912,-53.119,-178.141,6.037,148.529
C09976=1206.616,149.162,-53.141,-178.139,6.039,148.529
C09977=1206.611,149.411,-53.162,-178.137,6.040,148.529
C09978=1206.606,149.660,-53.183,-178.133,6.041,148.528
C09979=1206.601,149.909,-53.204,-178.131,6.043,148.528
C09980=1206.596,150.158,-53.225,-178.129,6.044,148.527
C09981=1206.592,150.407,-53.246,-178.126,6.046,148.527
C09982=1206.587,150.657,-53.267,-178.123,6.047,148.526
C09983=1206.582,150.905,-53.289,-178.121,6.048,148.526
C09984=1206.578,151.154,-53.309,-178.118,6.050,148.525
C09985=1206.573,151.403,-53.330,-178.115,6.052,148.525
C09986=1206.568,151.652,-53.352,-178.113,6.052,148.524
C09987=1206.563,151.902,-53.373,-178.110,6.054,148.524
C09988=1206.559,152.150,-53.394,-178.108,6.055,148.524
C09989=1206.554,152.400,-53.415,-178.105,6.057,148.523
C09990=1206.549,152.648,-53.437,-178.102,6.059,148.523
C09991=1206.545,152.898,-53.458,-178.100,6.059,148.522
C09992=1206.540,153.146,-53.479,-178.097,6.061,148.522
C09993=1206.535,153.396,-53.500,-178.094,6.063,148.521
C09994=1206.530,153.644,-53.522,-178.092,6.064,148.521
C09995=1206.525,153.894,-53.543,-178.089,6.065,148.521
C09996=1206.522,154.143,-53.564,-178.087,6.067,148.520
//INST
///DATE 2021/06/25 14:27
///ATTR SC,RW,RJ
////FRAME ROBOT
///GROUP1 RB1
NOP
MOVL C00000 V=800.0 PL=0
MOVL C00001 V=800.0 PL=0
MOVL C00002 V=800.0 PL=0
MOVL C00003 V=800.0 PL=0
MOVL C00004 V=800.0 PL=0
MOVL C00005 V=800.0 PL=0
MOVL C00006 V=800.0 PL=0
MOVL C00007 V=800.0 PL=0
MOVL C00008 V=800.0 PL=0
MOVL C00009 V=800.0 PL=0
MOVL C00010 V=800.0 PL=0
MOVL C00011 V=800.0 PL=0
MOVL C00012 V=800.0 PL=0
MOVL C00013 V=800.0 PL=0
MOVL C00014 V=800.0 PL=0
MOVL C00015 V=800.0 PL=0
MOVL C00016 V=800.0 PL=0
MOVL C00017 V=800.0 PL=0
MOVL C00018 V=800.0 PL=0
MOVL C00019 V=800.0 PL=0
MOVL C00020 V=800.0 PL=0
MOVL C00021 V=800.0 PL=0
MOVL C00022 V=800.0 PL=0
MOVL C00023 V=800.0 PL=0
MOVL C00024 V=800.0 PL=0
MOVL C00025 V=800.0 PL=0
MOVL C00026 V=800.0 PL=0
MOVL C00027 V=800.0 PL=0
MOVL C00028 V=800.0 PL=0
MOVL C00029 V=800.0 PL=0
MOVL C00030 V=800.0 PL=0
MOVL C00031 V=800.0 PL=0
MOVL C00032 V=800.0 PL=0
MOVL C00033 V=800.0 PL=0
MOVL C00034 V=800.0 PL=0
MOVL C00035 V=800.0 PL=0
MOVL C00036 V=800.0 PL=0
MOVL C00037 V=800.0 PL=0
MOVL C00038 V=800.0 PL=0
MOVL C00039 V=800.0 PL=0
MOVL C00040 V=800.0 PL=0
MOVL C00041 V=800.0 PL=0
MOVL C00042 V=800.0 PL=0
MOVL C00043 V=800.0 PL=0
MOVL C00044 V=800.0 PL=0
MOVL C00045 V=800.0 PL=0
MOVL C00046 V=800.0 PL=0
MOVL C00047 V=800.0 PL=0
MOVL C00048 V=800.0 PL=0
MOVL C00049 V=800.0 PL=0
MOVL C00050 V=800.0 PL=0
MOVL C00051 V=800.0 PL=0
MOVL C00052 V=800.0 PL=0
MOVL C00053 V=800.0 PL=0
MOVL C00054 V=800.0 PL=0
MOVL C00055 V=800.0 PL=0
MOVL C00056 V=800.0 PL=0
MOVL C00057 V=800.0 PL=0
MOVL C00058 V=800.0 PL=0
MOVL C00059 V=800.0 PL=0
MOVL C00060 V=800.0 PL=0
MOVL C00061 V=800.0 PL=0
MOVL C00062 V=800.0 PL=0
MOVL C00063 V=800.0 PL=0
MOVL C00064 V=800.0 PL=0
MOVL C00065 V=800.0 PL=0
MOVL C00066 V=800.0 PL=0
MOVL C00067 V=800.0 PL=0
MOVL C00068 V=800.0 PL=0
MOVL C00069 V=800.0 PL=0
MOVL C00070 V=800.0 PL=0
MOVL C00071 V=800.0 PL=0
MOVL C00072 V=800.0 PL=0
MOVL C00073 V=800.0 PL=0
MOVL C00074 V=800.0 PL=0
MOVL C00075 V=800.0 PL=0
MOVL C00076 V=800.0 PL=0
MOVL C00077 V=800.0 PL=0
MOVL C00078 V=800.0 PL=0
MOVL C00079 V=800.0 PL=0
MOVL C00080 V=800.0 PL=0
MOVL C00081 V=800.0 PL=0
MOVL C00082 V=800.0 PL=0
MOVL C00083 V=800.0 PL=0
MOVL C00084 V=800.0 PL=0
MOVL C00085 V=800.0 PL=0
MOVL C00086 V=800.0 PL=0
MOVL C00087 V=800.0 PL=0
MOVL C00088 V=800.0 PL=0
MOVL C00089 V=800.0 PL=0
MOVL C00090 V=800.0 PL=0
MOVL C00091 V=800.0 PL=0
MOVL C00092 V=800.0 PL=0
MOVL C00093 V=800.0 PL=0
MOVL C00094 V=800.0 PL=0
MOVL C00095 V=800.0 PL=0
MOVL C00096 V=800.0 PL=0
MOVL C00097 V=800.0 PL=0
MOVL C00098 V=800.0 PL=0
MOVL C00099 V=800.0 PL=0
MOVL C00100 V=800.0 PL=0
MOVL C00101 V=800.0 PL=0
MOVL C00102 V=800.0 PL=0
MOVL C00103 V=800.0 PL=0
MOVL C00104 V=800.0 PL=0
MOVL C00105 V=800.0 PL=0
MOVL C00106 V=800.0 PL=0
MOVL C00107 V=800.0 PL=0
MOVL C00108 V=800.0 PL=0
MOVL C00109 V=800.0 PL=0
MOVL C00110 V=800.0 PL=0
MOVL C00111 V=800.0 PL=0
MOVL C00112 V=800.0 PL=0
MOVL C00113 V=800.0 PL=0
MOVL C00114 V=800.0 PL=0
MOVL C00115 V=800.0 PL=0
MOVL C00116 V=800.0 PL=0
MOVL C00117 V=800.0 PL=0
MOVL C00118 V=800.0 PL=0
MOVL C00119 V=800.0 PL=0
MOVL C00120 V=800.0 PL=0
MOVL C00121 V=800.0 PL=0
MOVL C00122 V=800.0 PL=0
MOVL C00123 V=800.0 PL=0
MOVL C00124 V=800.0 PL=0
MOVL C00125 V=800.0 PL=0
MOVL C00126 V=800.0 PL=0
MOVL C00127 V=800.0 PL=0
MOVL C00128 V=800.0 PL=0
MOVL C00129 V=800.0 PL=0
MOVL C00130 V=800.0 PL=0
MOVL C00131 V=800.0 PL=0
MOVL C00132 V=800.0 PL=0
MOVL C00133 V=800.0 PL=0
MOVL C00134 V=800.0 PL=0
MOVL C00135 V=800.0 PL=0
MOVL C00136 V=800.0 PL=0
MOVL C00137 V=800.0 PL=0
MOVL C00138 V=800.0 PL=0
MOVL C00139 V=800.0 PL=0
MOVL C00140 V=800.0 PL=0
MOVL C00141 V=800.0 PL=0
MOVL C00142 V=800.0 PL=0
MOVL C00143 V=800.0 PL=0
MOVL C00144 V=800.0 PL=0
MOVL C00145 V=800.0 PL=0
MOVL C00146 V=800.0 PL=0
MOVL C00147 V=800.0 PL=0
MOVL C00148 V=800.0 PL=0
MOVL C00149 V=800.0 PL=0
MOVL C00150 V=800.0 PL=0
MOVL C00151 V=800.0 PL=0
MOVL C00152 V=800.0 PL=0
MOVL C00153 V=800.0 PL=0
MOVL C00154 V=800.0 PL=0
MOVL C00155 V=800.0 PL=0
MOVL C00156 V=800.0 PL=0
MOVL C00157 V=800.0 PL=0
MOVL C00158 V=800.0 PL=0
MOVL C00159 V=800.0 PL=0
MOVL C00160 V=800.0 PL=0
MOVL C00161 V=800.0 PL=0
MOVL C00162 V=800.0 PL=0
MOVL C00163 V=800.0 PL=0
MOVL C00164 V=800.0 PL=0
MOVL C00165 V=800.0 PL=0
MOVL C00166 V=800.0 PL=0
MOVL C00167 V=800.0 PL=0
MOVL C00168 V=800.0 PL=0
MOVL C00169 V=800.0 PL=0
MOVL C00170 V=800.0 PL=0
MOVL C00171 V=800.0 PL=0
MOVL C00172 V=800.0 PL=0
MOVL C00173 V=800.0 PL=0
MOVL C00174 V=800.0 PL=0
MOVL C00175 V=800.0 PL=0
MOVL C00176 V=800.0 PL=0
MOVL C00177 V=800.0 PL=0
MOVL C00178 V=800.0 PL=0
MOVL C00179 V=800.0 PL=0
MOVL C00180 V=800.0 PL=0
MOVL C00181 V=800.0 PL=0
MOVL C00182 V=800.0 PL=0
MOVL C00183 V=800.0 PL=0
MOVL C00184 V=800.0 PL=0
MOVL C00185 V=800.0 PL=0
MOVL C00186 V=800.0 PL=0
MOVL C00187 V=800.0 PL=0
MOVL C00188 V=800.0 PL=0
MOVL C00189 V=800.0 PL=0
MOVL C00190 V=800.0 PL=0
MOVL C00191 V=800.0 PL=0
MOVL C00192 V=800.0 PL=0
MOVL C00193 V=800.0 PL=0
MOVL C00194 V=800.0 PL=0
MOVL C00195 V=800.0 PL=0
MOVL C00196 V=800.0 PL=0
MOVL C00197 V=800.0 PL=0
MOVL C00198 V=800.0 PL=0
MOVL C00199 V=800.0 PL=0
MOVL C00200 V=800.0 PL=0
MOVL C00201 V=800.0 PL=0
MOVL C00202 V=800.0 PL=0
MOVL C00203 V=800.0 PL=0
MOVL C00204 V=800.0 PL=0
MOVL C00205 V=800.0 PL=0
MOVL C00206 V=800.0 PL=0
MOVL C00207 V=800.0 PL=0
MOVL C00208 V=800.0 PL=0
MOVL C00209 V=800.0 PL=0
MOVL C00210 V=800.0 PL=0
MOVL C00211 V=800.0 PL=0
MOVL C00212 V=800.0 PL=0
MOVL C00213 V=800.0 PL=0
MOVL C00214 V=800.0 PL=0
MOVL C00215 V=800.0 PL=0
MOVL C00216 V=800.0 PL=0
MOVL C00217 V=800.0 PL=0
MOVL C00218 V=800.0 PL=0
MOVL C00219 V=800.0 PL=0
MOVL C00220 V=800.0 PL=0
MOVL C00221 V=800.0 PL=0
MOVL C00222 V=800.0 PL=0
MOVL C00223 V=800.0 PL=0
MOVL C00224 V=800.0 PL=0
MOVL C00225 V=800.0 PL=0
MOVL C00226 V=800.0 PL=0
MOVL C00227 V=800.0 PL=0
MOVL C00228 V=800.0 PL=0
MOVL C00229 V=800.0 PL=0
MOVL C00230 V=800.0 PL=0
MOVL C00231 V=800.0 PL=0
MOVL C00232 V=800.0 PL=0
MOVL C00233 V=800.0 PL=0
MOVL C00234 V=800.0 PL=0
MOVL C00235 V=800.0 PL=0
MOVL C00236 V=800.0 PL=0
MOVL C00237 V=800.0 PL=0
MOVL C00238 V=800.0 PL=0
MOVL C00239 V=800.0 PL=0
MOVL C00240 V=800.0 PL=0
MOVL C00241 V=800.0 PL=0
MOVL C00242 V=800.0 PL=0
MOVL C00243 V=800.0 PL=0
MOVL C00244 V=800.0 PL=0
MOVL C00245 V=800.0 PL=0
MOVL C00246 V=800.0 PL=0
MOVL C00247 V=800.0 PL=0
MOVL C00248 V=800.0 PL=0
MOVL C00249 V=800.0 PL=0
MOVL C00250 V=800.0 PL=0
MOVL C00251 V=800.0 PL=0
MOVL C00252 V=800.0 PL=0
MOVL C00253 V=800.0 PL=0
MOVL C00254 V=800.0 PL=0
MOVL C00255 V=800.0 PL=0
MOVL C00256 V=800.0 PL=0
MOVL C00257 V=800.0 PL=0
MOVL C00258 V=800.0 PL=0
MOVL C00259 V=800.0 PL=0
MOVL C00260 V=800.0 PL=0
MOVL C00261 V=800.0 PL=0
MOVL C00262 V=800.0 PL=0
MOVL C00263 V=800.0 PL=0
MOVL C00264 V=800.0 PL=0
MOVL C00265 V=800.0 PL=0
MOVL C00266 V=800.0 PL=0
MOVL C00267 V=800.0 PL=0
MOVL C00268 V=800.0 PL=0
MOVL C00269 V=800.0 PL=0
MOVL C00270 V=800.0 PL=0
MOVL C00271 V=800.0 PL=0
MOVL C00272 V=800.0 PL=0
MOVL C00273 V=800.0 PL=0
MOVL C00274 V=800.0 PL=0
MOVL C00275 V=800.0 PL=0
MOVL C00276 V=800.0 PL=0
MOVL C00277 V=800.0 PL=0
MOVL C00278 V=800.0 PL=0
MOVL C00279 V=800.0 PL=0
MOVL C00280 V=800.0 PL=0
MOVL C00281 V=800.0 PL=0
MOVL C00282 V=800.0 PL=0
MOVL C00283 V=800.0 PL=0
MOVL C00284 V=800.0 PL=0
MOVL C00285 V=800.0 PL=0
MOVL C00286 V=800.0 PL=0
MOVL C00287 V=800.0 PL=0
MOVL C00288 V=800.0 PL=0
MOVL C00289 V=800.0 PL=0
MOVL C00290 V=800.0 PL=0
MOVL C00291 V=800.0 PL=0
MOVL C00292 V=800.0 PL=0
MOVL C00293 V=800.0 PL=0
MOVL C00294 V=800.0 PL=0
MOVL C00295 V=800.0 PL=0
MOVL C00296 V=800.0 PL=0
MOVL C00297 V=800.0 PL=0
MOVL C00298 V=800.0 PL=0
MOVL C00299 V=800.0 PL=0
MOVL C00300 V=800.0 PL=0
MOVL C00301 V=800.0 PL=0
MOVL C00302 V=800.0 PL=0
MOVL C00303 V=800.0 PL=0
MOVL C00304 V=800.0 PL=0
MOVL C00305 V=800.0 PL=0
MOVL C00306 V=800.0 PL=0
MOVL C00307 V=800.0 PL=0
MOVL C00308 V=800.0 PL=0
MOVL C00309 V=800.0 PL=0
MOVL C00310 V=800.0 PL=0
MOVL C00311 V=800.0 PL=0
MOVL C00312 V=800.0 PL=0
MOVL C00313 V=800.0 PL=0
MOVL C00314 V=800.0 PL=0
MOVL C00315 V=800.0 PL=0
MOVL C00316 V=800.0 PL=0
MOVL C00317 V=800.0 PL=0
MOVL C00318 V=800.0 PL=0
MOVL C00319 V=800.0 PL=0
MOVL C00320 V=800.0 PL=0
MOVL C00321 V=800.0 PL=0
MOVL C00322 V=800.0 PL=0
MOVL C00323 V=800.0 PL=0
MOVL C00324 V=800.0 PL=0
MOVL C00325 V=800.0 PL=0
MOVL C00326 V=800.0 PL=0
MOVL C00327 V=800.0 PL=0
MOVL C00328 V=800.0 PL=0
MOVL C00329 V=800.0 PL=0
MOVL C00330 V=800.0 PL=0
MOVL C00331 V=800.0 PL=0
MOVL C00332 V=800.0 PL=0
MOVL C00333 V=800.0 PL=0
MOVL C00334 V=800.0 PL=0
MOVL C00335 V=800.0 PL=0
MOVL C00336 V=800.0 PL=0
MOVL C00337 V=800.0 PL=0
MOVL C00338 V=800.0 PL=0
MOVL C00339 V=800.0 PL=0
MOVL C00340 V=800.0 PL=0
MOVL C00341 V=800.0 PL=0
MOVL C00342 V=800.0 PL=0
MOVL C00343 V=800.0 PL=0
MOVL C00344 V=800.0 PL=0
MOVL C00345 V=800.0 PL=0
MOVL C00346 V=800.0 PL=0
MOVL C00347 V=800.0 PL=0
MOVL C00348 V=800.0 PL=0
MOVL C00349 V=800.0 PL=0
MOVL C00350 V=800.0 PL=0
MOVL C00351 V=800.0 PL=0
MOVL C00352 V=800.0 PL=0
MOVL C00353 V=800.0 PL=0
MOVL C00354 V=800.0 PL=0
MOVL C00355 V=800.0 PL=0
MOVL C00356 V=800.0 PL=0
MOVL C00357 V=800.0 PL=0
MOVL C00358 V=800.0 PL=0
MOVL C00359 V=800.0 PL=0
MOVL C00360 V=800.0 PL=0
MOVL C00361 V=800.0 PL=0
MOVL C00362 V=800.0 PL=0
MOVL C00363 V=800.0 PL=0
MOVL C00364 V=800.0 PL=0
MOVL C00365 V=800.0 PL=0
MOVL C00366 V=800.0 PL=0
MOVL C00367 V=800.0 PL=0
MOVL C00368 V=800.0 PL=0
MOVL C00369 V=800.0 PL=0
MOVL C00370 V=800.0 PL=0
MOVL C00371 V=800.0 PL=0
MOVL C00372 V=800.0 PL=0
MOVL C00373 V=800.0 PL=0
MOVL C00374 V=800.0 PL=0
MOVL C00375 V=800.0 PL=0
MOVL C00376 V=800.0 PL=0
MOVL C00377 V=800.0 PL=0
MOVL C00378 V=800.0 PL=0
MOVL C00379 V=800.0 PL=0
MOVL C00380 V=800.0 PL=0
MOVL C00381 V=800.0 PL=0
MOVL C00382 V=800.0 PL=0
MOVL C00383 V=800.0 PL=0
MOVL C00384 V=800.0 PL=0
MOVL C00385 V=800.0 PL=0
MOVL C00386 V=800.0 PL=0
MOVL C00387 V=800.0 PL=0
MOVL C00388 V=800.0 PL=0
MOVL C00389 V=800.0 PL=0
MOVL C00390 V=800.0 PL=0
MOVL C00391 V=800.0 PL=0
MOVL C00392 V=800.0 PL=0
MOVL C00393 V=800.0 PL=0
MOVL C00394 V=800.0 PL=0
MOVL C00395 V=800.0 PL=0
MOVL C00396 V=800.0 PL=0
MOVL C00397 V=800.0 PL=0
MOVL C00398 V=800.0 PL=0
MOVL C00399 V=800.0 PL=0
MOVL C00400 V=800.0 PL=0
MOVL C00401 V=800.0 PL=0
MOVL C00402 V=800.0 PL=0
MOVL C00403 V=800.0 PL=0
MOVL C00404 V=800.0 PL=0
MOVL C00405 V=800.0 PL=0
MOVL C00406 V=800.0 PL=0
MOVL C00407 V=800.0 PL=0
MOVL C00408 V=800.0 PL=0
MOVL C00409 V=800.0 PL=0
MOVL C00410 V=800.0 PL=0
MOVL C00411 V=800.0 PL=0
MOVL C00412 V=800.0 PL=0
MOVL C00413 V=800.0 PL=0
MOVL C00414 V=800.0 PL=0
MOVL C00415 V=800.0 PL=0
MOVL C00416 V=800.0 PL=0
MOVL C00417 V=800.0 PL=0
MOVL C00418 V=800.0 PL=0
MOVL C00419 V=800.0 PL=0
MOVL C00420 V=800.0 PL=0
MOVL C00421 V=800.0 PL=0
MOVL C00422 V=800.0 PL=0
MOVL C00423 V=800.0 PL=0
MOVL C00424 V=800.0 PL=0
MOVL C00425 V=800.0 PL=0
MOVL C00426 V=800.0 PL=0
MOVL C00427 V=800.0 PL=0
MOVL C00428 V=800.0 PL=0
MOVL C00429 V=800.0 PL=0
MOVL C00430 V=800.0 PL=0
MOVL C00431 V=800.0 PL=0
MOVL C00432 V=800.0 PL=0
MOVL C00433 V=800.0 PL=0
MOVL C00434 V=800.0 PL=0
MOVL C00435 V=800.0 PL=0
MOVL C00436 V=800.0 PL=0
MOVL C00437 V=800.0 PL=0
MOVL C00438 V=800.0 PL=0
MOVL C00439 V=800.0 PL=0
MOVL C00440 V=800.0 PL=0
MOVL C00441 V=800.0 PL=0
MOVL C00442 V=800.0 PL=0
MOVL C00443 V=800.0 PL=0
MOVL C00444 V=800.0 PL=0
MOVL C00445 V=800.0 PL=0
MOVL C00446 V=800.0 PL=0
MOVL C00447 V=800.0 PL=0
MOVL C00448 V=800.0 PL=0
MOVL C00449 V=800.0 PL=0
MOVL C00450 V=800.0 PL=0
MOVL C00451 V=800.0 PL=0
MOVL C00452 V=800.0 PL=0
MOVL C00453 V=800.0 PL=0
MOVL C00454 V=800.0 PL=0
MOVL C00455 V=800.0 PL=0
MOVL C00456 V=800.0 PL=0
MOVL C00457 V=800.0 PL=0
MOVL C00458 V=800.0 PL=0
MOVL C00459 V=800.0 PL=0
MOVL C00460 V=800.0 PL=0
MOVL C00461 V=800.0 PL=0
MOVL C00462 V=800.0 PL=0
MOVL C00463 V=800.0 PL=0
MOVL C00464 V=800.0 PL=0
MOVL C00465 V=800.0 PL=0
MOVL C00466 V=800.0 PL=0
MOVL C00467 V=800.0 PL=0
MOVL C00468 V=800.0 PL=0
MOVL C00469 V=800.0 PL=0
MOVL C00470 V=800.0 PL=0
MOVL C00471 V=800.0 PL=0
MOVL C00472 V=800.0 PL=0
MOVL C00473 V=800.0 PL=0
MOVL C00474 V=800.0 PL=0
MOVL C00475 V=800.0 PL=0
MOVL C00476 V=800.0 PL=0
MOVL C00477 V=800.0 PL=0
MOVL C00478 V=800.0 PL=0
MOVL C00479 V=800.0 PL=0
MOVL C00480 V=800.0 PL=0
MOVL C00481 V=800.0 PL=0
MOVL C00482 V=800.0 PL=0
MOVL C00483 V=800.0 PL=0
MOVL C00484 V=800.0 PL=0
MOVL C00485 V=800.0 PL=0
MOVL C00486 V=800.0 PL=0
MOVL C00487 V=800.0 PL=0
MOVL C00488 V=800.0 PL=0
MOVL C00489 V=800.0 PL=0
MOVL C00490 V=800.0 PL=0
MOVL C00491 V=800.0 PL=0
MOVL C00492 V=800.0 PL=0
MOVL C00493 V=800.0 PL=0
MOVL C00494 V=800.0 PL=0
MOVL C00495 V=800.0 PL=0
MOVL C00496 V=800.0 PL=0
MOVL C00497 V=800.0 PL=0
MOVL C00498 V=800.0 PL=0
MOVL C00499 V=800.0 PL=0
MOVL C00500 V=800.0 PL=0
MOVL C00501 V=800.0 PL=0
MOVL C00502 V=800.0 PL=0
MOVL C00503 V=800.0 PL=0
MOVL C00504 V=800.0 PL=0
MOVL C00505 V=800.0 PL=0
MOVL C00506 V=800.0 PL=0
MOVL C00507 V=800.0 PL=0
MOVL C00508 V=800.0 PL=0
MOVL C00509 V=800.0 PL=0
MOVL C00510 V=800.0 PL=0
MOVL C00511 V=800.0 PL=0
MOVL C00512 V=800.0 PL=0
MOVL C00513 V=800.0 PL=0
MOVL C00514 V=800.0 PL=0
MOVL C00515 V=800.0 PL=0
MOVL C00516 V=800.0 PL=0
MOVL C00517 V=800.0 PL=0
MOVL C00518 V=800.0 PL=0
MOVL C00519 V=800.0 PL=0
MOVL C00520 V=800.0 PL=0
MOVL C00521 V=800.0 PL=0
MOVL C00522 V=800.0 PL=0
MOVL C00523 V=800.0 PL=0
MOVL C00524 V=800.0 PL=0
MOVL C00525 V=800.0 PL=0
MOVL C00526 V=800.0 PL=0
MOVL C00527 V=800.0 PL=0
MOVL C00528 V=800.0 PL=0
MOVL C00529 V=800.0 PL=0
MOVL C00530 V=800.0 PL=0
MOVL C00531 V=800.0 PL=0
MOVL C00532 V=800.0 PL=0
MOVL C00533 V=800.0 PL=0
MOVL C00534 V=800.0 PL=0
MOVL C00535 V=800.0 PL=0
MOVL C00536 V=800.0 PL=0
MOVL C00537 V=800.0 PL=0
MOVL C00538 V=800.0 PL=0
MOVL C00539 V=800.0 PL=0
MOVL C00540 V=800.0 PL=0
MOVL C00541 V=800.0 PL=0
MOVL C00542 V=800.0 PL=0
MOVL C00543 V=800.0 PL=0
MOVL C00544 V=800.0 PL=0
MOVL C00545 V=800.0 PL=0
MOVL C00546 V=800.0 PL=0
MOVL C00547 V=800.0 PL=0
MOVL C00548 V=800.0 PL=0
MOVL C00549 V=800.0 PL=0
MOVL C00550 V=800.0 PL=0
MOVL C00551 V=800.0 PL=0
MOVL C00552 V=800.0 PL=0
MOVL C00553 V=800.0 PL=0
MOVL C00554 V=800.0 PL=0
MOVL C00555 V=800.0 PL=0
MOVL C00556 V=800.0 PL=0
MOVL C00557 V=800.0 PL=0
MOVL C00558 V=800.0 PL=0
MOVL C00559 V=800.0 PL=0
MOVL C00560 V=800.0 PL=0
MOVL C00561 V=800.0 PL=0
MOVL C00562 V=800.0 PL=0
MOVL C00563 V=800.0 PL=0
MOVL C00564 V=800.0 PL=0
MOVL C00565 V=800.0 PL=0
MOVL C00566 V=800.0 PL=0
MOVL C00567 V=800.0 PL=0
MOVL C00568 V=800.0 PL=0
MOVL C00569 V=800.0 PL=0
MOVL C00570 V=800.0 PL=0
MOVL C00571 V=800.0 PL=0
MOVL C00572 V=800.0 PL=0
MOVL C00573 V=800.0 PL=0
MOVL C00574 V=800.0 PL=0
MOVL C00575 V=800.0 PL=0
MOVL C00576 V=800.0 PL=0
MOVL C00577 V=800.0 PL=0
MOVL C00578 V=800.0 PL=0
MOVL C00579 V=800.0 PL=0
MOVL C00580 V=800.0 PL=0
MOVL C00581 V=800.0 PL=0
MOVL C00582 V=800.0 PL=0
MOVL C00583 V=800.0 PL=0
MOVL C00584 V=800.0 PL=0
MOVL C00585 V=800.0 PL=0
MOVL C00586 V=800.0 PL=0
MOVL C00587 V=800.0 PL=0
MOVL C00588 V=800.0 PL=0
MOVL C00589 V=800.0 PL=0
MOVL C00590 V=800.0 PL=0
MOVL C00591 V=800.0 PL=0
MOVL C00592 V=800.0 PL=0
MOVL C00593 V=800.0 PL=0
MOVL C00594 V=800.0 PL=0
MOVL C00595 V=800.0 PL=0
MOVL C00596 V=800.0 PL=0
MOVL C00597 V=800.0 PL=0
MOVL C00598 V=800.0 PL=0
MOVL C00599 V=800.0 PL=0
MOVL C00600 V=800.0 PL=0
MOVL C00601 V=800.0 PL=0
MOVL C00602 V=800.0 PL=0
MOVL C00603 V=800.0 PL=0
MOVL C00604 V=800.0 PL=0
MOVL C00605 V=800.0 PL=0
MOVL C00606 V=800.0 PL=0
MOVL C00607 V=800.0 PL=0
MOVL C00608 V=800.0 PL=0
MOVL C00609 V=800.0 PL=0
MOVL C00610 V=800.0 PL=0
MOVL C00611 V=800.0 PL=0
MOVL C00612 V=800.0 PL=0
MOVL C00613 V=800.0 PL=0
MOVL C00614 V=800.0 PL=0
MOVL C00615 V=800.0 PL=0
MOVL C00616 V=800.0 PL=0
MOVL C00617 V=800.0 PL=0
MOVL C00618 V=800.0 PL=0
MOVL C00619 V=800.0 PL=0
MOVL C00620 V=800.0 PL=0
MOVL C00621 V=800.0 PL=0
MOVL C00622 V=800.0 PL=0
MOVL C00623 V=800.0 PL=0
MOVL C00624 V=800.0 PL=0
MOVL C00625 V=800.0 PL=0
MOVL C00626 V=800.0 PL=0
MOVL C00627 V=800.0 PL=0
MOVL C00628 V=800.0 PL=0
MOVL C00629 V=800.0 PL=0
MOVL C00630 V=800.0 PL=0
MOVL C00631 V=800.0 PL=0
MOVL C00632 V=800.0 PL=0
MOVL C00633 V=800.0 PL=0
MOVL C00634 V=800.0 PL=0
MOVL C00635 V=800.0 PL=0
MOVL C00636 V=800.0 PL=0
MOVL C00637 V=800.0 PL=0
MOVL C00638 V=800.0 PL=0
MOVL C00639 V=800.0 PL=0
MOVL C00640 V=800.0 PL=0
MOVL C00641 V=800.0 PL=0
MOVL C00642 V=800.0 PL=0
MOVL C00643 V=800.0 PL=0
MOVL C00644 V=800.0 PL=0
MOVL C00645 V=800.0 PL=0
MOVL C00646 V=800.0 PL=0
MOVL C00647 V=800.0 PL=0
MOVL C00648 V=800.0 PL=0
MOVL C00649 V=800.0 PL=0
MOVL C00650 V=800.0 PL=0
MOVL C00651 V=800.0 PL=0
MOVL C00652 V=800.0 PL=0
MOVL C00653 V=800.0 PL=0
MOVL C00654 V=800.0 PL=0
MOVL C00655 V=800.0 PL=0
MOVL C00656 V=800.0 PL=0
MOVL C00657 V=800.0 PL=0
MOVL C00658 V=800.0 PL=0
MOVL C00659 V=800.0 PL=0
MOVL C00660 V=800.0 PL=0
MOVL C00661 V=800.0 PL=0
MOVL C00662 V=800.0 PL=0
MOVL C00663 V=800.0 PL=0
MOVL C00664 V=800.0 PL=0
MOVL C00665 V=800.0 PL=0
MOVL C00666 V=800.0 PL=0
MOVL C00667 V=800.0 PL=0
MOVL C00668 V=800.0 PL=0
MOVL C00669 V=800.0 PL=0
MOVL C00670 V=800.0 PL=0
MOVL C00671 V=800.0 PL=0
MOVL C00672 V=800.0 PL=0
MOVL C00673 V=800.0 PL=0
MOVL C00674 V=800.0 PL=0
MOVL C00675 V=800.0 PL=0
MOVL C00676 V=800.0 PL=0
MOVL C00677 V=800.0 PL=0
MOVL C00678 V=800.0 PL=0
MOVL C00679 V=800.0 PL=0
MOVL C00680 V=800.0 PL=0
MOVL C00681 V=800.0 PL=0
MOVL C00682 V=800.0 PL=0
MOVL C00683 V=800.0 PL=0
MOVL C00684 V=800.0 PL=0
MOVL C00685 V=800.0 PL=0
MOVL C00686 V=800.0 PL=0
MOVL C00687 V=800.0 PL=0
MOVL C00688 V=800.0 PL=0
MOVL C00689 V=800.0 PL=0
MOVL C00690 V=800.0 PL=0
MOVL C00691 V=800.0 PL=0
MOVL C00692 V=800.0 PL=0
MOVL C00693 V=800.0 PL=0
MOVL C00694 V=800.0 PL=0
MOVL C00695 V=800.0 PL=0
MOVL C00696 V=800.0 PL=0
MOVL C00697 V=800.0 PL=0
MOVL C00698 V=800.0 PL=0
MOVL C00699 V=800.0 PL=0
MOVL C00700 V=800.0 PL=0
MOVL C00701 V=800.0 PL=0
MOVL C00702 V=800.0 PL=0
MOVL C00703 V=800.0 PL=0
MOVL C00704 V=800.0 PL=0
MOVL C00705 V=800.0 PL=0
MOVL C00706 V=800.0 PL=0
MOVL C00707 V=800.0 PL=0
MOVL C00708 V=800.0 PL=0
MOVL C00709 V=800.0 PL=0
MOVL C00710 V=800.0 PL=0
MOVL C00711 V=800.0 PL=0
MOVL C00712 V=800.0 PL=0
MOVL C00713 V=800.0 PL=0
MOVL C00714 V=800.0 PL=0
MOVL C00715 V=800.0 PL=0
MOVL C00716 V=800.0 PL=0
MOVL C00717 V=800.0 PL=0
MOVL C00718 V=800.0 PL=0
MOVL C00719 V=800.0 PL=0
MOVL C00720 V=800.0 PL=0
MOVL C00721 V=800.0 PL=0
MOVL C00722 V=800.0 PL=0
MOVL C00723 V=800.0 PL=0
MOVL C00724 V=800.0 PL=0
MOVL C00725 V=800.0 PL=0
MOVL C00726 V=800.0 PL=0
MOVL C00727 V=800.0 PL=0
MOVL C00728 V=800.0 PL=0
MOVL C00729 V=800.0 PL=0
MOVL C00730 V=800.0 PL=0
MOVL C00731 V=800.0 PL=0
MOVL C00732 V=800.0 PL=0
MOVL C00733 V=800.0 PL=0
MOVL C00734 V=800.0 PL=0
MOVL C00735 V=800.0 PL=0
MOVL C00736 V=800.0 PL=0
MOVL C00737 V=800.0 PL=0
MOVL C00738 V=800.0 PL=0
MOVL C00739 V=800.0 PL=0
MOVL C00740 V=800.0 PL=0
MOVL C00741 V=800.0 PL=0
MOVL C00742 V=800.0 PL=0
MOVL C00743 V=800.0 PL=0
MOVL C00744 V=800.0 PL=0
MOVL C00745 V=800.0 PL=0
MOVL C00746 V=800.0 PL=0
MOVL C00747 V=800.0 PL=0
MOVL C00748 V=800.0 PL=0
MOVL C00749 V=800.0 PL=0
MOVL C00750 V=800.0 PL=0
MOVL C00751 V=800.0 PL=0
MOVL C00752 V=800.0 PL=0
MOVL C00753 V=800.0 PL=0
MOVL C00754 V=800.0 PL=0
MOVL C00755 V=800.0 PL=0
MOVL C00756 V=800.0 PL=0
MOVL C00757 V=800.0 PL=0
MOVL C00758 V=800.0 PL=0
MOVL C00759 V=800.0 PL=0
MOVL C00760 V=800.0 PL=0
MOVL C00761 V=800.0 PL=0
MOVL C00762 V=800.0 PL=0
MOVL C00763 V=800.0 PL=0
MOVL C00764 V=800.0 PL=0
MOVL C00765 V=800.0 PL=0
MOVL C00766 V=800.0 PL=0
MOVL C00767 V=800.0 PL=0
MOVL C00768 V=800.0 PL=0
MOVL C00769 V=800.0 PL=0
MOVL C00770 V=800.0 PL=0
MOVL C00771 V=800.0 PL=0
MOVL C00772 V=800.0 PL=0
MOVL C00773 V=800.0 PL=0
MOVL C00774 V=800.0 PL=0
MOVL C00775 V=800.0 PL=0
MOVL C00776 V=800.0 PL=0
MOVL C00777 V=800.0 PL=0
MOVL C00778 V=800.0 PL=0
MOVL C00779 V=800.0 PL=0
MOVL C00780 V=800.0 PL=0
MOVL C00781 V=800.0 PL=0
MOVL C00782 V=800.0 PL=0
MOVL C00783 V=800.0 PL=0
MOVL C00784 V=800.0 PL=0
MOVL C00785 V=800.0 PL=0
MOVL C00786 V=800.0 PL=0
MOVL C00787 V=800.0 PL=0
MOVL C00788 V=800.0 PL=0
MOVL C00789 V=800.0 PL=0
MOVL C00790 V=800.0 PL=0
MOVL C00791 V=800.0 PL=0
MOVL C00792 V=800.0 PL=0
MOVL C00793 V=800.0 PL=0
MOVL C00794 V=800.0 PL=0
MOVL C00795 V=800.0 PL=0
MOVL C00796 V=800.0 PL=0
MOVL C00797 V=800.0 PL=0
MOVL C00798 V=800.0 PL=0
MOVL C00799 V=800.0 PL=0
MOVL C00800 V=800.0 PL=0
MOVL C00801 V=800.0 PL=0
MOVL C00802 V=800.0 PL=0
MOVL C00803 V=800.0 PL=0
MOVL C00804 V=800.0 PL=0
MOVL C00805 V=800.0 PL=0
MOVL C00806 V=800.0 PL=0
MOVL C00807 V=800.0 PL=0
MOVL C00808 V=800.0 PL=0
MOVL C00809 V=800.0 PL=0
MOVL C00810 V=800.0 PL=0
MOVL C00811 V=800.0 PL=0
MOVL C00812 V=800.0 PL=0
MOVL C00813 V=800.0 PL=0
MOVL C00814 V=800.0 PL=0
MOVL C00815 V=800.0 PL=0
MOVL C00816 V=800.0 PL=0
MOVL C00817 V=800.0 PL=0
MOVL C00818 V=800.0 PL=0
MOVL C00819 V=800.0 PL=0
MOVL C00820 V=800.0 PL=0
MOVL C00821 V=800.0 PL=0
MOVL C00822 V=800.0 PL=0
MOVL C00823 V=800.0 PL=0
MOVL C00824 V=800.0 PL=0
MOVL C00825 V=800.0 PL=0
MOVL C00826 V=800.0 PL=0
MOVL C00827 V=800.0 PL=0
MOVL C00828 V=800.0 PL=0
MOVL C00829 V=800.0 PL=0
MOVL C00830 V=800.0 PL=0
MOVL C00831 V=800.0 PL=0
MOVL C00832 V=800.0 PL=0
MOVL C00833 V=800.0 PL=0
MOVL C00834 V=800.0 PL=0
MOVL C00835 V=800.0 PL=0
MOVL C00836 V=800.0 PL=0
MOVL C00837 V=800.0 PL=0
MOVL C00838 V=800.0 PL=0
MOVL C00839 V=800.0 PL=0
MOVL C00840 V=800.0 PL=0
MOVL C00841 V=800.0 PL=0
MOVL C00842 V=800.0 PL=0
MOVL C00843 V=800.0 PL=0
MOVL C00844 V=800.0 PL=0
MOVL C00845 V=800.0 PL=0
MOVL C00846 V=800.0 PL=0
MOVL C00847 V=800.0 PL=0
MOVL C00848 V=800.0 PL=0
MOVL C00849 V=800.0 PL=0
MOVL C00850 V=800.0 PL=0
MOVL C00851 V=800.0 PL=0
MOVL C00852 V=800.0 PL=0
MOVL C00853 V=800.0 PL=0
MOVL C00854 V=800.0 PL=0
MOVL C00855 V=800.0 PL=0
MOVL C00856 V=800.0 PL=0
MOVL C00857 V=800.0 PL=0
MOVL C00858 V=800.0 PL=0
MOVL C00859 V=800.0 PL=0
MOVL C00860 V=800.0 PL=0
MOVL C00861 V=800.0 PL=0
MOVL C00862 V=800.0 PL=0
MOVL C00863 V=800.0 PL=0
MOVL C00864 V=800.0 PL=0
MOVL C00865 V=800.0 PL=0
MOVL C00866 V=800.0 PL=0
MOVL C00867 V=800.0 PL=0
MOVL C00868 V=800.0 PL=0
MOVL C00869 V=800.0 PL=0
MOVL C00870 V=800.0 PL=0
MOVL C00871 V=800.0 PL=0
MOVL C00872 V=800.0 PL=0
MOVL C00873 V=800.0 PL=0
MOVL C00874 V=800.0 PL=0
MOVL C00875 V=800.0 PL=0
MOVL C00876 V=800.0 PL=0
MOVL C00877 V=800.0 PL=0
MOVL C00878 V=800.0 PL=0
MOVL C00879 V=800.0 PL=0
MOVL C00880 V=800.0 PL=0
MOVL C00881 V=800.0 PL=0
MOVL C00882 V=800.0 PL=0
MOVL C00883 V=800.0 PL=0
MOVL C00884 V=800.0 PL=0
MOVL C00885 V=800.0 PL=0
MOVL C00886 V=800.0 PL=0
MOVL C00887 V=800.0 PL=0
MOVL C00888 V=800.0 PL=0
MOVL C00889 V=800.0 PL=0
MOVL C00890 V=800.0 PL=0
MOVL C00891 V=800.0 PL=0
MOVL C00892 V=800.0 PL=0
MOVL C00893 V=800.0 PL=0
MOVL C00894 V=800.0 PL=0
MOVL C00895 V=800.0 PL=0
MOVL C00896 V=800.0 PL=0
MOVL C00897 V=800.0 PL=0
MOVL C00898 V=800.0 PL=0
MOVL C00899 V=800.0 PL=0
MOVL C00900 V=800.0 PL=0
MOVL C00901 V=800.0 PL=0
MOVL C00902 V=800.0 PL=0
MOVL C00903 V=800.0 PL=0
MOVL C00904 V=800.0 PL=0
MOVL C00905 V=800.0 PL=0
MOVL C00906 V=800.0 PL=0
MOVL C00907 V=800.0 PL=0
MOVL C00908 V=800.0 PL=0
MOVL C00909 V=800.0 PL=0
MOVL C00910 V=800.0 PL=0
MOVL C00911 V=800.0 PL=0
MOVL C00912 V=800.0 PL=0
MOVL C00913 V=800.0 PL=0
MOVL C00914 V=800.0 PL=0
MOVL C00915 V=800.0 PL=0
MOVL C00916 V=800.0 PL=0
MOVL C00917 V=800.0 PL=0
MOVL C00918 V=800.0 PL=0
MOVL C00919 V=800.0 PL=0
MOVL C00920 V=800.0 PL=0
MOVL C00921 V=800.0 PL=0
MOVL C00922 V=800.0 PL=0
MOVL C00923 V=800.0 PL=0
MOVL C00924 V=800.0 PL=0
MOVL C00925 V=800.0 PL=0
MOVL C00926 V=800.0 PL=0
MOVL C00927 V=800.0 PL=0
MOVL C00928 V=800.0 PL=0
MOVL C00929 V=800.0 PL=0
MOVL C00930 V=800.0 PL=0
MOVL C00931 V=800.0 PL=0
MOVL C00932 V=800.0 PL=0
MOVL C00933 V=800.0 PL=0
MOVL C00934 V=800.0 PL=0
MOVL C00935 V=800.0 PL=0
MOVL C00936 V=800.0 PL=0
MOVL C00937 V=800.0 PL=0
MOVL C00938 V=800.0 PL=0
MOVL C00939 V=800.0 PL=0
MOVL C00940 V=800.0 PL=0
MOVL C00941 V=800.0 PL=0
MOVL C00942 V=800.0 PL=0
MOVL C00943 V=800.0 PL=0
MOVL C00944 V=800.0 PL=0
MOVL C00945 V=800.0 PL=0
MOVL C00946 V=800.0 PL=0
MOVL C00947 V=800.0 PL=0
MOVL C00948 V=800.0 PL=0
MOVL C00949 V=800.0 PL=0
MOVL C00950 V=800.0 PL=0
MOVL C00951 V=800.0 PL=0
MOVL C00952 V=800.0 PL=0
MOVL C00953 V=800.0 PL=0
MOVL C00954 V=800.0 PL=0
MOVL C00955 V=800.0 PL=0
MOVL C00956 V=800.0 PL=0
MOVL C00957 V=800.0 PL=0
MOVL C00958 V=800.0 PL=0
MOVL C00959 V=800.0 PL=0
MOVL C00960 V=800.0 PL=0
MOVL C00961 V=800.0 PL=0
MOVL C00962 V=800.0 PL=0
MOVL C00963 V=800.0 PL=0
MOVL C00964 V=800.0 PL=0
MOVL C00965 V=800.0 PL=0
MOVL C00966 V=800.0 PL=0
MOVL C00967 V=800.0 PL=0
MOVL C00968 V=800.0 PL=0
MOVL C00969 V=800.0 PL=0
MOVL C00970 V=800.0 PL=0
MOVL C00971 V=800.0 PL=0
MOVL C00972 V=800.0 PL=0
MOVL C00973 V=800.0 PL=0
MOVL C00974 V=800.0 PL=0
MOVL C00975 V=800.0 PL=0
MOVL C00976 V=800.0 PL=0
MOVL C00977 V=800.0 PL=0
MOVL C00978 V=800.0 PL=0
MOVL C00979 V=800.0 PL=0
MOVL C00980 V=800.0 PL=0
MOVL C00981 V=800.0 PL=0
MOVL C00982 V=800.0 PL=0
MOVL C00983 V=800.0 PL=0
MOVL C00984 V=800.0 PL=0
MOVL C00985 V=800.0 PL=0
MOVL C00986 V=800.0 PL=0
MOVL C00987 V=800.0 PL=0
MOVL C00988 V=800.0 PL=0
MOVL C00989 V=800.0 PL=0
MOVL C00990 V=800.0 PL=0
MOVL C00991 V=800.0 PL=0
MOVL C00992 V=800.0 PL=0
MOVL C00993 V=800.0 PL=0
MOVL C00994 V=800.0 PL=0
MOVL C00995 V=800.0 PL=0
MOVL C00996 V=800.0 PL=0
MOVL C00997 V=800.0 PL=0
MOVL C00998 V=800.0 PL=0
MOVL C00999 V=800.0 PL=0
MOVL C01000 V=800.0 PL=0
MOVL C01001 V=800.0 PL=0
MOVL C01002 V=800.0 PL=0
MOVL C01003 V=800.0 PL=0
MOVL C01004 V=800.0 PL=0
MOVL C01005 V=800.0 PL=0
MOVL C01006 V=800.0 PL=0
MOVL C01007 V=800.0 PL=0
MOVL C01008 V=800.0 PL=0
MOVL C01009 V=800.0 PL=0
MOVL C01010 V=800.0 PL=0
MOVL C01011 V=800.0 PL=0
MOVL C01012 V=800.0 PL=0
MOVL C01013 V=800.0 PL=0
MOVL C01014 V=800.0 PL=0
MOVL C01015 V=800.0 PL=0
MOVL C01016 V=800.0 PL=0
MOVL C01017 V=800.0 PL=0
MOVL C01018 V=800.0 PL=0
MOVL C01019 V=800.0 PL=0
MOVL C01020 V=800.0 PL=0
MOVL C01021 V=800.0 PL=0
MOVL C01022 V=800.0 PL=0
MOVL C01023 V=800.0 PL=0
MOVL C01024 V=800.0 PL=0
MOVL C01025 V=800.0 PL=0
MOVL C01026 V=800.0 PL=0
MOVL C01027 V=800.0 PL=0
MOVL C01028 V=800.0 PL=0
MOVL C01029 V=800.0 PL=0
MOVL C01030 V=800.0 PL=0
MOVL C01031 V=800.0 PL=0
MOVL C01032 V=800.0 PL=0
MOVL C01033 V=800.0 PL=0
MOVL C01034 V=800.0 PL=0
MOVL C01035 V=800.0 PL=0
MOVL C01036 V=800.0 PL=0
MOVL C01037 V=800.0 PL=0
MOVL C01038 V=800.0 PL=0
MOVL C01039 V=800.0 PL=0
MOVL C01040 V=800.0 PL=0
MOVL C01041 V=800.0 PL=0
MOVL C01042 V=800.0 PL=0
MOVL C01043 V=800.0 PL=0
MOVL C01044 V=800.0 PL=0
MOVL C01045 V=800.0 PL=0
MOVL C01046 V=800.0 PL=0
MOVL C01047 V=800.0 PL=0
MOVL C01048 V=800.0 PL=0
MOVL C01049 V=800.0 PL=0
MOVL C01050 V=800.0 PL=0
MOVL C01051 V=800.0 PL=0
MOVL C01052 V=800.0 PL=0
MOVL C01053 V=800.0 PL=0
MOVL C01054 V=800.0 PL=0
MOVL C01055 V=800.0 PL=0
MOVL C01056 V=800.0 PL=0
MOVL C01057 V=800.0 PL=0
MOVL C01058 V=800.0 PL=0
MOVL C01059 V=800.0 PL=0
MOVL C01060 V=800.0 PL=0
MOVL C01061 V=800.0 PL=0
MOVL C01062 V=800.0 PL=0
MOVL C01063 V=800.0 PL=0
MOVL C01064 V=800.0 PL=0
MOVL C01065 V=800.0 PL=0
MOVL C01066 V=800.0 PL=0
MOVL C01067 V=800.0 PL=0
MOVL C01068 V=800.0 PL=0
MOVL C01069 V=800.0 PL=0
MOVL C01070 V=800.0 PL=0
MOVL C01071 V=800.0 PL=0
MOVL C01072 V=800.0 PL=0
MOVL C01073 V=800.0 PL=0
MOVL C01074 V=800.0 PL=0
MOVL C01075 V=800.0 PL=0
MOVL C01076 V=800.0 PL=0
MOVL C01077 V=800.0 PL=0
MOVL C01078 V=800.0 PL=0
MOVL C01079 V=800.0 PL=0
MOVL C01080 V=800.0 PL=0
MOVL C01081 V=800.0 PL=0
MOVL C01082 V=800.0 PL=0
MOVL C01083 V=800.0 PL=0
MOVL C01084 V=800.0 PL=0
MOVL C01085 V=800.0 PL=0
MOVL C01086 V=800.0 PL=0
MOVL C01087 V=800.0 PL=0
MOVL C01088 V=800.0 PL=0
MOVL C01089 V=800.0 PL=0
MOVL C01090 V=800.0 PL=0
MOVL C01091 V=800.0 PL=0
MOVL C01092 V=800.0 PL=0
MOVL C01093 V=800.0 PL=0
MOVL C01094 V=800.0 PL=0
MOVL C01095 V=800.0 PL=0
MOVL C01096 V=800.0 PL=0
MOVL C01097 V=800.0 PL=0
MOVL C01098 V=800.0 PL=0
MOVL C01099 V=800.0 PL=0
MOVL C01100 V=800.0 PL=0
MOVL C01101 V=800.0 PL=0
MOVL C01102 V=800.0 PL=0
MOVL C01103 V=800.0 PL=0
MOVL C01104 V=800.0 PL=0
MOVL C01105 V=800.0 PL=0
MOVL C01106 V=800.0 PL=0
MOVL C01107 V=800.0 PL=0
MOVL C01108 V=800.0 PL=0
MOVL C01109 V=800.0 PL=0
MOVL C01110 V=800.0 PL=0
MOVL C01111 V=800.0 PL=0
MOVL C01112 V=800.0 PL=0
MOVL C01113 V=800.0 PL=0
MOVL C01114 V=800.0 PL=0
MOVL C01115 V=800.0 PL=0
MOVL C01116 V=800.0 PL=0
MOVL C01117 V=800.0 PL=0
MOVL C01118 V=800.0 PL=0
MOVL C01119 V=800.0 PL=0
MOVL C01120 V=800.0 PL=0
MOVL C01121 V=800.0 PL=0
MOVL C01122 V=800.0 PL=0
MOVL C01123 V=800.0 PL=0
MOVL C01124 V=800.0 PL=0
MOVL C01125 V=800.0 PL=0
MOVL C01126 V=800.0 PL=0
MOVL C01127 V=800.0 PL=0
MOVL C01128 V=800.0 PL=0
MOVL C01129 V=800.0 PL=0
MOVL C01130 V=800.0 PL=0
MOVL C01131 V=800.0 PL=0
MOVL C01132 V=800.0 PL=0
MOVL C01133 V=800.0 PL=0
MOVL C01134 V=800.0 PL=0
MOVL C01135 V=800.0 PL=0
MOVL C01136 V=800.0 PL=0
MOVL C01137 V=800.0 PL=0
MOVL C01138 V=800.0 PL=0
MOVL C01139 V=800.0 PL=0
MOVL C01140 V=800.0 PL=0
MOVL C01141 V=800.0 PL=0
MOVL C01142 V=800.0 PL=0
MOVL C01143 V=800.0 PL=0
MOVL C01144 V=800.0 PL=0
MOVL C01145 V=800.0 PL=0
MOVL C01146 V=800.0 PL=0
MOVL C01147 V=800.0 PL=0
MOVL C01148 V=800.0 PL=0
MOVL C01149 V=800.0 PL=0
MOVL C01150 V=800.0 PL=0
MOVL C01151 V=800.0 PL=0
MOVL C01152 V=800.0 PL=0
MOVL C01153 V=800.0 PL=0
MOVL C01154 V=800.0 PL=0
MOVL C01155 V=800.0 PL=0
MOVL C01156 V=800.0 PL=0
MOVL C01157 V=800.0 PL=0
MOVL C01158 V=800.0 PL=0
MOVL C01159 V=800.0 PL=0
MOVL C01160 V=800.0 PL=0
MOVL C01161 V=800.0 PL=0
MOVL C01162 V=800.0 PL=0
MOVL C01163 V=800.0 PL=0
MOVL C01164 V=800.0 PL=0
MOVL C01165 V=800.0 PL=0
MOVL C01166 V=800.0 PL=0
MOVL C01167 V=800.0 PL=0
MOVL C01168 V=800.0 PL=0
MOVL C01169 V=800.0 PL=0
MOVL C01170 V=800.0 PL=0
MOVL C01171 V=800.0 PL=0
MOVL C01172 V=800.0 PL=0
MOVL C01173 V=800.0 PL=0
MOVL C01174 V=800.0 PL=0
MOVL C01175 V=800.0 PL=0
MOVL C01176 V=800.0 PL=0
MOVL C01177 V=800.0 PL=0
MOVL C01178 V=800.0 PL=0
MOVL C01179 V=800.0 PL=0
MOVL C01180 V=800.0 PL=0
MOVL C01181 V=800.0 PL=0
MOVL C01182 V=800.0 PL=0
MOVL C01183 V=800.0 PL=0
MOVL C01184 V=800.0 PL=0
MOVL C01185 V=800.0 PL=0
MOVL C01186 V=800.0 PL=0
MOVL C01187 V=800.0 PL=0
MOVL C01188 V=800.0 PL=0
MOVL C01189 V=800.0 PL=0
MOVL C01190 V=800.0 PL=0
MOVL C01191 V=800.0 PL=0
MOVL C01192 V=800.0 PL=0
MOVL C01193 V=800.0 PL=0
MOVL C01194 V=800.0 PL=0
MOVL C01195 V=800.0 PL=0
MOVL C01196 V=800.0 PL=0
MOVL C01197 V=800.0 PL=0
MOVL C01198 V=800.0 PL=0
MOVL C01199 V=800.0 PL=0
MOVL C01200 V=800.0 PL=0
MOVL C01201 V=800.0 PL=0
MOVL C01202 V=800.0 PL=0
MOVL C01203 V=800.0 PL=0
MOVL C01204 V=800.0 PL=0
MOVL C01205 V=800.0 PL=0
MOVL C01206 V=800.0 PL=0
MOVL C01207 V=800.0 PL=0
MOVL C01208 V=800.0 PL=0
MOVL C01209 V=800.0 PL=0
MOVL C01210 V=800.0 PL=0
MOVL C01211 V=800.0 PL=0
MOVL C01212 V=800.0 PL=0
MOVL C01213 V=800.0 PL=0
MOVL C01214 V=800.0 PL=0
MOVL C01215 V=800.0 PL=0
MOVL C01216 V=800.0 PL=0
MOVL C01217 V=800.0 PL=0
MOVL C01218 V=800.0 PL=0
MOVL C01219 V=800.0 PL=0
MOVL C01220 V=800.0 PL=0
MOVL C01221 V=800.0 PL=0
MOVL C01222 V=800.0 PL=0
MOVL C01223 V=800.0 PL=0
MOVL C01224 V=800.0 PL=0
MOVL C01225 V=800.0 PL=0
MOVL C01226 V=800.0 PL=0
MOVL C01227 V=800.0 PL=0
MOVL C01228 V=800.0 PL=0
MOVL C01229 V=800.0 PL=0
MOVL C01230 V=800.0 PL=0
MOVL C01231 V=800.0 PL=0
MOVL C01232 V=800.0 PL=0
MOVL C01233 V=800.0 PL=0
MOVL C01234 V=800.0 PL=0
MOVL C01235 V=800.0 PL=0
MOVL C01236 V=800.0 PL=0
MOVL C01237 V=800.0 PL=0
MOVL C01238 V=800.0 PL=0
MOVL C01239 V=800.0 PL=0
MOVL C01240 V=800.0 PL=0
MOVL C01241 V=800.0 PL=0
MOVL C01242 V=800.0 PL=0
MOVL C01243 V=800.0 PL=0
MOVL C01244 V=800.0 PL=0
MOVL C01245 V=800.0 PL=0
MOVL C01246 V=800.0 PL=0
MOVL C01247 V=800.0 PL=0
MOVL C01248 V=800.0 PL=0
MOVL C01249 V=800.0 PL=0
MOVL C01250 V=800.0 PL=0
MOVL C01251 V=800.0 PL=0
MOVL C01252 V=800.0 PL=0
MOVL C01253 V=800.0 PL=0
MOVL C01254 V=800.0 PL=0
MOVL C01255 V=800.0 PL=0
MOVL C01256 V=800.0 PL=0
MOVL C01257 V=800.0 PL=0
MOVL C01258 V=800.0 PL=0
MOVL C01259 V=800.0 PL=0
MOVL C01260 V=800.0 PL=0
MOVL C01261 V=800.0 PL=0
MOVL C01262 V=800.0 PL=0
MOVL C01263 V=800.0 PL=0
MOVL C01264 V=800.0 PL=0
MOVL C01265 V=800.0 PL=0
MOVL C01266 V=800.0 PL=0
MOVL C01267 V=800.0 PL=0
MOVL C01268 V=800.0 PL=0
MOVL C01269 V=800.0 PL=0
MOVL C01270 V=800.0 PL=0
MOVL C01271 V=800.0 PL=0
MOVL C01272 V=800.0 PL=0
MOVL C01273 V=800.0 PL=0
MOVL C01274 V=800.0 PL=0
MOVL C01275 V=800.0 PL=0
MOVL C01276 V=800.0 PL=0
MOVL C01277 V=800.0 PL=0
MOVL C01278 V=800.0 PL=0
MOVL C01279 V=800.0 PL=0
MOVL C01280 V=800.0 PL=0
MOVL C01281 V=800.0 PL=0
MOVL C01282 V=800.0 PL=0
MOVL C01283 V=800.0 PL=0
MOVL C01284 V=800.0 PL=0
MOVL C01285 V=800.0 PL=0
MOVL C01286 V=800.0 PL=0
MOVL C01287 V=800.0 PL=0
MOVL C01288 V=800.0 PL=0
MOVL C01289 V=800.0 PL=0
MOVL C01290 V=800.0 PL=0
MOVL C01291 V=800.0 PL=0
MOVL C01292 V=800.0 PL=0
MOVL C01293 V=800.0 PL=0
MOVL C01294 V=800.0 PL=0
MOVL C01295 V=800.0 PL=0
MOVL C01296 V=800.0 PL=0
MOVL C01297 V=800.0 PL=0
MOVL C01298 V=800.0 PL=0
MOVL C01299 V=800.0 PL=0
MOVL C01300 V=800.0 PL=0
MOVL C01301 V=800.0 PL=0
MOVL C01302 V=800.0 PL=0
MOVL C01303 V=800.0 PL=0
MOVL C01304 V=800.0 PL=0
MOVL C01305 V=800.0 PL=0
MOVL C01306 V=800.0 PL=0
MOVL C01307 V=800.0 PL=0
MOVL C01308 V=800.0 PL=0
MOVL C01309 V=800.0 PL=0
MOVL C01310 V=800.0 PL=0
MOVL C01311 V=800.0 PL=0
MOVL C01312 V=800.0 PL=0
MOVL C01313 V=800.0 PL=0
MOVL C01314 V=800.0 PL=0
MOVL C01315 V=800.0 PL=0
MOVL C01316 V=800.0 PL=0
MOVL C01317 V=800.0 PL=0
MOVL C01318 V=800.0 PL=0
MOVL C01319 V=800.0 PL=0
MOVL C01320 V=800.0 PL=0
MOVL C01321 V=800.0 PL=0
MOVL C01322 V=800.0 PL=0
MOVL C01323 V=800.0 PL=0
MOVL C01324 V=800.0 PL=0
MOVL C01325 V=800.0 PL=0
MOVL C01326 V=800.0 PL=0
MOVL C01327 V=800.0 PL=0
MOVL C01328 V=800.0 PL=0
MOVL C01329 V=800.0 PL=0
MOVL C01330 V=800.0 PL=0
MOVL C01331 V=800.0 PL=0
MOVL C01332 V=800.0 PL=0
MOVL C01333 V=800.0 PL=0
MOVL C01334 V=800.0 PL=0
MOVL C01335 V=800.0 PL=0
MOVL C01336 V=800.0 PL=0
MOVL C01337 V=800.0 PL=0
MOVL C01338 V=800.0 PL=0
MOVL C01339 V=800.0 PL=0
MOVL C01340 V=800.0 PL=0
MOVL C01341 V=800.0 PL=0
MOVL C01342 V=800.0 PL=0
MOVL C01343 V=800.0 PL=0
MOVL C01344 V=800.0 PL=0
MOVL C01345 V=800.0 PL=0
MOVL C01346 V=800.0 PL=0
MOVL C01347 V=800.0 PL=0
MOVL C01348 V=800.0 PL=0
MOVL C01349 V=800.0 PL=0
MOVL C01350 V=800.0 PL=0
MOVL C01351 V=800.0 PL=0
MOVL C01352 V=800.0 PL=0
MOVL C01353 V=800.0 PL=0
MOVL C01354 V=800.0 PL=0
MOVL C01355 V=800.0 PL=0
MOVL C01356 V=800.0 PL=0
MOVL C01357 V=800.0 PL=0
MOVL C01358 V=800.0 PL=0
MOVL C01359 V=800.0 PL=0
MOVL C01360 V=800.0 PL=0
MOVL C01361 V=800.0 PL=0
MOVL C01362 V=800.0 PL=0
MOVL C01363 V=800.0 PL=0
MOVL C01364 V=800.0 PL=0
MOVL C01365 V=800.0 PL=0
MOVL C01366 V=800.0 PL=0
MOVL C01367 V=800.0 PL=0
MOVL C01368 V=800.0 PL=0
MOVL C01369 V=800.0 PL=0
MOVL C01370 V=800.0 PL=0
MOVL C01371 V=800.0 PL=0
MOVL C01372 V=800.0 PL=0
MOVL C01373 V=800.0 PL=0
MOVL C01374 V=800.0 PL=0
MOVL C01375 V=800.0 PL=0
MOVL C01376 V=800.0 PL=0
MOVL C01377 V=800.0 PL=0
MOVL C01378 V=800.0 PL=0
MOVL C01379 V=800.0 PL=0
MOVL C01380 V=800.0 PL=0
MOVL C01381 V=800.0 PL=0
MOVL C01382 V=800.0 PL=0
MOVL C01383 V=800.0 PL=0
MOVL C01384 V=800.0 PL=0
MOVL C01385 V=800.0 PL=0
MOVL C01386 V=800.0 PL=0
MOVL C01387 V=800.0 PL=0
MOVL C01388 V=800.0 PL=0
MOVL C01389 V=800.0 PL=0
MOVL C01390 V=800.0 PL=0
MOVL C01391 V=800.0 PL=0
MOVL C01392 V=800.0 PL=0
MOVL C01393 V=800.0 PL=0
MOVL C01394 V=800.0 PL=0
MOVL C01395 V=800.0 PL=0
MOVL C01396 V=800.0 PL=0
MOVL C01397 V=800.0 PL=0
MOVL C01398 V=800.0 PL=0
MOVL C01399 V=800.0 PL=0
MOVL C01400 V=800.0 PL=0
MOVL C01401 V=800.0 PL=0
MOVL C01402 V=800.0 PL=0
MOVL C01403 V=800.0 PL=0
MOVL C01404 V=800.0 PL=0
MOVL C01405 V=800.0 PL=0
MOVL C01406 V=800.0 PL=0
MOVL C01407 V=800.0 PL=0
MOVL C01408 V=800.0 PL=0
MOVL C01409 V=800.0 PL=0
MOVL C01410 V=800.0 PL=0
MOVL C01411 V=800.0 PL=0
MOVL C01412 V=800.0 PL=0
MOVL C01413 V=800.0 PL=0
MOVL C01414 V=800.0 PL=0
MOVL C01415 V=800.0 PL=0
MOVL C01416 V=800.0 PL=0
MOVL C01417 V=800.0 PL=0
MOVL C01418 V=800.0 PL=0
MOVL C01419 V=800.0 PL=0
MOVL C01420 V=800.0 PL=0
MOVL C01421 V=800.0 PL=0
MOVL C01422 V=800.0 PL=0
MOVL C01423 V=800.0 PL=0
MOVL C01424 V=800.0 PL=0
MOVL C01425 V=800.0 PL=0
MOVL C01426 V=800.0 PL=0
MOVL C01427 V=800.0 PL=0
MOVL C01428 V=800.0 PL=0
MOVL C01429 V=800.0 PL=0
MOVL C01430 V=800.0 PL=0
MOVL C01431 V=800.0 PL=0
MOVL C01432 V=800.0 PL=0
MOVL C01433 V=800.0 PL=0
MOVL C01434 V=800.0 PL=0
MOVL C01435 V=800.0 PL=0
MOVL C01436 V=800.0 PL=0
MOVL C01437 V=800.0 PL=0
MOVL C01438 V=800.0 PL=0
MOVL C01439 V=800.0 PL=0
MOVL C01440 V=800.0 PL=0
MOVL C01441 V=800.0 PL=0
MOVL C01442 V=800.0 PL=0
MOVL C01443 V=800.0 PL=0
MOVL C01444 V=800.0 PL=0
MOVL C01445 V=800.0 PL=0
MOVL C01446 V=800.0 PL=0
MOVL C01447 V=800.0 PL=0
MOVL C01448 V=800.0 PL=0
MOVL C01449 V=800.0 PL=0
MOVL C01450 V=800.0 PL=0
MOVL C01451 V=800.0 PL=0
MOVL C01452 V=800.0 PL=0
MOVL C01453 V=800.0 PL=0
MOVL C01454 V=800.0 PL=0
MOVL C01455 V=800.0 PL=0
MOVL C01456 V=800.0 PL=0
MOVL C01457 V=800.0 PL=0
MOVL C01458 V=800.0 PL=0
MOVL C01459 V=800.0 PL=0
MOVL C01460 V=800.0 PL=0
MOVL C01461 V=800.0 PL=0
MOVL C01462 V=800.0 PL=0
MOVL C01463 V=800.0 PL=0
MOVL C01464 V=800.0 PL=0
MOVL C01465 V=800.0 PL=0
MOVL C01466 V=800.0 PL=0
MOVL C01467 V=800.0 PL=0
MOVL C01468 V=800.0 PL=0
MOVL C01469 V=800.0 PL=0
MOVL C01470 V=800.0 PL=0
MOVL C01471 V=800.0 PL=0
MOVL C01472 V=800.0 PL=0
MOVL C01473 V=800.0 PL=0
MOVL C01474 V=800.0 PL=0
MOVL C01475 V=800.0 PL=0
MOVL C01476 V=800.0 PL=0
MOVL C01477 V=800.0 PL=0
MOVL C01478 V=800.0 PL=0
MOVL C01479 V=800.0 PL=0
MOVL C01480 V=800.0 PL=0
MOVL C01481 V=800.0 PL=0
MOVL C01482 V=800.0 PL=0
MOVL C01483 V=800.0 PL=0
MOVL C01484 V=800.0 PL=0
MOVL C01485 V=800.0 PL=0
MOVL C01486 V=800.0 PL=0
MOVL C01487 V=800.0 PL=0
MOVL C01488 V=800.0 PL=0
MOVL C01489 V=800.0 PL=0
MOVL C01490 V=800.0 PL=0
MOVL C01491 V=800.0 PL=0
MOVL C01492 V=800.0 PL=0
MOVL C01493 V=800.0 PL=0
MOVL C01494 V=800.0 PL=0
MOVL C01495 V=800.0 PL=0
MOVL C01496 V=800.0 PL=0
MOVL C01497 V=800.0 PL=0
MOVL C01498 V=800.0 PL=0
MOVL C01499 V=800.0 PL=0
MOVL C01500 V=800.0 PL=0
MOVL C01501 V=800.0 PL=0
MOVL C01502 V=800.0 PL=0
MOVL C01503 V=800.0 PL=0
MOVL C01504 V=800.0 PL=0
MOVL C01505 V=800.0 PL=0
MOVL C01506 V=800.0 PL=0
MOVL C01507 V=800.0 PL=0
MOVL C01508 V=800.0 PL=0
MOVL C01509 V=800.0 PL=0
MOVL C01510 V=800.0 PL=0
MOVL C01511 V=800.0 PL=0
MOVL C01512 V=800.0 PL=0
MOVL C01513 V=800.0 PL=0
MOVL C01514 V=800.0 PL=0
MOVL C01515 V=800.0 PL=0
MOVL C01516 V=800.0 PL=0
MOVL C01517 V=800.0 PL=0
MOVL C01518 V=800.0 PL=0
MOVL C01519 V=800.0 PL=0
MOVL C01520 V=800.0 PL=0
MOVL C01521 V=800.0 PL=0
MOVL C01522 V=800.0 PL=0
MOVL C01523 V=800.0 PL=0
MOVL C01524 V=800.0 PL=0
MOVL C01525 V=800.0 PL=0
MOVL C01526 V=800.0 PL=0
MOVL C01527 V=800.0 PL=0
MOVL C01528 V=800.0 PL=0
MOVL C01529 V=800.0 PL=0
MOVL C01530 V=800.0 PL=0
MOVL C01531 V=800.0 PL=0
MOVL C01532 V=800.0 PL=0
MOVL C01533 V=800.0 PL=0
MOVL C01534 V=800.0 PL=0
MOVL C01535 V=800.0 PL=0
MOVL C01536 V=800.0 PL=0
MOVL C01537 V=800.0 PL=0
MOVL C01538 V=800.0 PL=0
MOVL C01539 V=800.0 PL=0
MOVL C01540 V=800.0 PL=0
MOVL C01541 V=800.0 PL=0
MOVL C01542 V=800.0 PL=0
MOVL C01543 V=800.0 PL=0
MOVL C01544 V=800.0 PL=0
MOVL C01545 V=800.0 PL=0
MOVL C01546 V=800.0 PL=0
MOVL C01547 V=800.0 PL=0
MOVL C01548 V=800.0 PL=0
MOVL C01549 V=800.0 PL=0
MOVL C01550 V=800.0 PL=0
MOVL C01551 V=800.0 PL=0
MOVL C01552 V=800.0 PL=0
MOVL C01553 V=800.0 PL=0
MOVL C01554 V=800.0 PL=0
MOVL C01555 V=800.0 PL=0
MOVL C01556 V=800.0 PL=0
MOVL C01557 V=800.0 PL=0
MOVL C01558 V=800.0 PL=0
MOVL C01559 V=800.0 PL=0
MOVL C01560 V=800.0 PL=0
MOVL C01561 V=800.0 PL=0
MOVL C01562 V=800.0 PL=0
MOVL C01563 V=800.0 PL=0
MOVL C01564 V=800.0 PL=0
MOVL C01565 V=800.0 PL=0
MOVL C01566 V=800.0 PL=0
MOVL C01567 V=800.0 PL=0
MOVL C01568 V=800.0 PL=0
MOVL C01569 V=800.0 PL=0
MOVL C01570 V=800.0 PL=0
MOVL C01571 V=800.0 PL=0
MOVL C01572 V=800.0 PL=0
MOVL C01573 V=800.0 PL=0
MOVL C01574 V=800.0 PL=0
MOVL C01575 V=800.0 PL=0
MOVL C01576 V=800.0 PL=0
MOVL C01577 V=800.0 PL=0
MOVL C01578 V=800.0 PL=0
MOVL C01579 V=800.0 PL=0
MOVL C01580 V=800.0 PL=0
MOVL C01581 V=800.0 PL=0
MOVL C01582 V=800.0 PL=0
MOVL C01583 V=800.0 PL=0
MOVL C01584 V=800.0 PL=0
MOVL C01585 V=800.0 PL=0
MOVL C01586 V=800.0 PL=0
MOVL C01587 V=800.0 PL=0
MOVL C01588 V=800.0 PL=0
MOVL C01589 V=800.0 PL=0
MOVL C01590 V=800.0 PL=0
MOVL C01591 V=800.0 PL=0
MOVL C01592 V=800.0 PL=0
MOVL C01593 V=800.0 PL=0
MOVL C01594 V=800.0 PL=0
MOVL C01595 V=800.0 PL=0
MOVL C01596 V=800.0 PL=0
MOVL C01597 V=800.0 PL=0
MOVL C01598 V=800.0 PL=0
MOVL C01599 V=800.0 PL=0
MOVL C01600 V=800.0 PL=0
MOVL C01601 V=800.0 PL=0
MOVL C01602 V=800.0 PL=0
MOVL C01603 V=800.0 PL=0
MOVL C01604 V=800.0 PL=0
MOVL C01605 V=800.0 PL=0
MOVL C01606 V=800.0 PL=0
MOVL C01607 V=800.0 PL=0
MOVL C01608 V=800.0 PL=0
MOVL C01609 V=800.0 PL=0
MOVL C01610 V=800.0 PL=0
MOVL C01611 V=800.0 PL=0
MOVL C01612 V=800.0 PL=0
MOVL C01613 V=800.0 PL=0
MOVL C01614 V=800.0 PL=0
MOVL C01615 V=800.0 PL=0
MOVL C01616 V=800.0 PL=0
MOVL C01617 V=800.0 PL=0
MOVL C01618 V=800.0 PL=0
MOVL C01619 V=800.0 PL=0
MOVL C01620 V=800.0 PL=0
MOVL C01621 V=800.0 PL=0
MOVL C01622 V=800.0 PL=0
MOVL C01623 V=800.0 PL=0
MOVL C01624 V=800.0 PL=0
MOVL C01625 V=800.0 PL=0
MOVL C01626 V=800.0 PL=0
MOVL C01627 V=800.0 PL=0
MOVL C01628 V=800.0 PL=0
MOVL C01629 V=800.0 PL=0
MOVL C01630 V=800.0 PL=0
MOVL C01631 V=800.0 PL=0
MOVL C01632 V=800.0 PL=0
MOVL C01633 V=800.0 PL=0
MOVL C01634 V=800.0 PL=0
MOVL C01635 V=800.0 PL=0
MOVL C01636 V=800.0 PL=0
MOVL C01637 V=800.0 PL=0
MOVL C01638 V=800.0 PL=0
MOVL C01639 V=800.0 PL=0
MOVL C01640 V=800.0 PL=0
MOVL C01641 V=800.0 PL=0
MOVL C01642 V=800.0 PL=0
MOVL C01643 V=800.0 PL=0
MOVL C01644 V=800.0 PL=0
MOVL C01645 V=800.0 PL=0
MOVL C01646 V=800.0 PL=0
MOVL C01647 V=800.0 PL=0
MOVL C01648 V=800.0 PL=0
MOVL C01649 V=800.0 PL=0
MOVL C01650 V=800.0 PL=0
MOVL C01651 V=800.0 PL=0
MOVL C01652 V=800.0 PL=0
MOVL C01653 V=800.0 PL=0
MOVL C01654 V=800.0 PL=0
MOVL C01655 V=800.0 PL=0
MOVL C01656 V=800.0 PL=0
MOVL C01657 V=800.0 PL=0
MOVL C01658 V=800.0 PL=0
MOVL C01659 V=800.0 PL=0
MOVL C01660 V=800.0 PL=0
MOVL C01661 V=800.0 PL=0
MOVL C01662 V=800.0 PL=0
MOVL C01663 V=800.0 PL=0
MOVL C01664 V=800.0 PL=0
MOVL C01665 V=800.0 PL=0
MOVL C01666 V=800.0 PL=0
MOVL C01667 V=800.0 PL=0
MOVL C01668 V=800.0 PL=0
MOVL C01669 V=800.0 PL=0
MOVL C01670 V=800.0 PL=0
MOVL C01671 V=800.0 PL=0
MOVL C01672 V=800.0 PL=0
MOVL C01673 V=800.0 PL=0
MOVL C01674 V=800.0 PL=0
MOVL C01675 V=800.0 PL=0
MOVL C01676 V=800.0 PL=0
MOVL C01677 V=800.0 PL=0
MOVL C01678 V=800.0 PL=0
MOVL C01679 V=800.0 PL=0
MOVL C01680 V=800.0 PL=0
MOVL C01681 V=800.0 PL=0
MOVL C01682 V=800.0 PL=0
MOVL C01683 V=800.0 PL=0
MOVL C01684 V=800.0 PL=0
MOVL C01685 V=800.0 PL=0
MOVL C01686 V=800.0 PL=0
MOVL C01687 V=800.0 PL=0
MOVL C01688 V=800.0 PL=0
MOVL C01689 V=800.0 PL=0
MOVL C01690 V=800.0 PL=0
MOVL C01691 V=800.0 PL=0
MOVL C01692 V=800.0 PL=0
MOVL C01693 V=800.0 PL=0
MOVL C01694 V=800.0 PL=0
MOVL C01695 V=800.0 PL=0
MOVL C01696 V=800.0 PL=0
MOVL C01697 V=800.0 PL=0
MOVL C01698 V=800.0 PL=0
MOVL C01699 V=800.0 PL=0
MOVL C01700 V=800.0 PL=0
MOVL C01701 V=800.0 PL=0
MOVL C01702 V=800.0 PL=0
MOVL C01703 V=800.0 PL=0
MOVL C01704 V=800.0 PL=0
MOVL C01705 V=800.0 PL=0
MOVL C01706 V=800.0 PL=0
MOVL C01707 V=800.0 PL=0
MOVL C01708 V=800.0 PL=0
MOVL C01709 V=800.0 PL=0
MOVL C01710 V=800.0 PL=0
MOVL C01711 V=800.0 PL=0
MOVL C01712 V=800.0 PL=0
MOVL C01713 V=800.0 PL=0
MOVL C01714 V=800.0 PL=0
MOVL C01715 V=800.0 PL=0
MOVL C01716 V=800.0 PL=0
MOVL C01717 V=800.0 PL=0
MOVL C01718 V=800.0 PL=0
MOVL C01719 V=800.0 PL=0
MOVL C01720 V=800.0 PL=0
MOVL C01721 V=800.0 PL=0
MOVL C01722 V=800.0 PL=0
MOVL C01723 V=800.0 PL=0
MOVL C01724 V=800.0 PL=0
MOVL C01725 V=800.0 PL=0
MOVL C01726 V=800.0 PL=0
MOVL C01727 V=800.0 PL=0
MOVL C01728 V=800.0 PL=0
MOVL C01729 V=800.0 PL=0
MOVL C01730 V=800.0 PL=0
MOVL C01731 V=800.0 PL=0
MOVL C01732 V=800.0 PL=0
MOVL C01733 V=800.0 PL=0
MOVL C01734 V=800.0 PL=0
MOVL C01735 V=800.0 PL=0
MOVL C01736 V=800.0 PL=0
MOVL C01737 V=800.0 PL=0
MOVL C01738 V=800.0 PL=0
MOVL C01739 V=800.0 PL=0
MOVL C01740 V=800.0 PL=0
MOVL C01741 V=800.0 PL=0
MOVL C01742 V=800.0 PL=0
MOVL C01743 V=800.0 PL=0
MOVL C01744 V=800.0 PL=0
MOVL C01745 V=800.0 PL=0
MOVL C01746 V=800.0 PL=0
MOVL C01747 V=800.0 PL=0
MOVL C01748 V=800.0 PL=0
MOVL C01749 V=800.0 PL=0
MOVL C01750 V=800.0 PL=0
MOVL C01751 V=800.0 PL=0
MOVL C01752 V=800.0 PL=0
MOVL C01753 V=800.0 PL=0
MOVL C01754 V=800.0 PL=0
MOVL C01755 V=800.0 PL=0
MOVL C01756 V=800.0 PL=0
MOVL C01757 V=800.0 PL=0
MOVL C01758 V=800.0 PL=0
MOVL C01759 V=800.0 PL=0
MOVL C01760 V=800.0 PL=0
MOVL C01761 V=800.0 PL=0
MOVL C01762 V=800.0 PL=0
MOVL C01763 V=800.0 PL=0
MOVL C01764 V=800.0 PL=0
MOVL C01765 V=800.0 PL=0
MOVL C01766 V=800.0 PL=0
MOVL C01767 V=800.0 PL=0
MOVL C01768 V=800.0 PL=0
MOVL C01769 V=800.0 PL=0
MOVL C01770 V=800.0 PL=0
MOVL C01771 V=800.0 PL=0
MOVL C01772 V=800.0 PL=0
MOVL C01773 V=800.0 PL=0
MOVL C01774 V=800.0 PL=0
MOVL C01775 V=800.0 PL=0
MOVL C01776 V=800.0 PL=0
MOVL C01777 V=800.0 PL=0
MOVL C01778 V=800.0 PL=0
MOVL C01779 V=800.0 PL=0
MOVL C01780 V=800.0 PL=0
MOVL C01781 V=800.0 PL=0
MOVL C01782 V=800.0 PL=0
MOVL C01783 V=800.0 PL=0
MOVL C01784 V=800.0 PL=0
MOVL C01785 V=800.0 PL=0
MOVL C01786 V=800.0 PL=0
MOVL C01787 V=800.0 PL=0
MOVL C01788 V=800.0 PL=0
MOVL C01789 V=800.0 PL=0
MOVL C01790 V=800.0 PL=0
MOVL C01791 V=800.0 PL=0
MOVL C01792 V=800.0 PL=0
MOVL C01793 V=800.0 PL=0
MOVL C01794 V=800.0 PL=0
MOVL C01795 V=800.0 PL=0
MOVL C01796 V=800.0 PL=0
MOVL C01797 V=800.0 PL=0
MOVL C01798 V=800.0 PL=0
MOVL C01799 V=800.0 PL=0
MOVL C01800 V=800.0 PL=0
MOVL C01801 V=800.0 PL=0
MOVL C01802 V=800.0 PL=0
MOVL C01803 V=800.0 PL=0
MOVL C01804 V=800.0 PL=0
MOVL C01805 V=800.0 PL=0
MOVL C01806 V=800.0 PL=0
MOVL C01807 V=800.0 PL=0
MOVL C01808 V=800.0 PL=0
MOVL C01809 V=800.0 PL=0
MOVL C01810 V=800.0 PL=0
MOVL C01811 V=800.0 PL=0
MOVL C01812 V=800.0 PL=0
MOVL C01813 V=800.0 PL=0
MOVL C01814 V=800.0 PL=0
MOVL C01815 V=800.0 PL=0
MOVL C01816 V=800.0 PL=0
MOVL C01817 V=800.0 PL=0
MOVL C01818 V=800.0 PL=0
MOVL C01819 V=800.0 PL=0
MOVL C01820 V=800.0 PL=0
MOVL C01821 V=800.0 PL=0
MOVL C01822 V=800.0 PL=0
MOVL C01823 V=800.0 PL=0
MOVL C01824 V=800.0 PL=0
MOVL C01825 V=800.0 PL=0
MOVL C01826 V=800.0 PL=0
MOVL C01827 V=800.0 PL=0
MOVL C01828 V=800.0 PL=0
MOVL C01829 V=800.0 PL=0
MOVL C01830 V=800.0 PL=0
MOVL C01831 V=800.0 PL=0
MOVL C01832 V=800.0 PL=0
MOVL C01833 V=800.0 PL=0
MOVL C01834 V=800.0 PL=0
MOVL C01835 V=800.0 PL=0
MOVL C01836 V=800.0 PL=0
MOVL C01837 V=800.0 PL=0
MOVL C01838 V=800.0 PL=0
MOVL C01839 V=800.0 PL=0
MOVL C01840 V=800.0 PL=0
MOVL C01841 V=800.0 PL=0
MOVL C01842 V=800.0 PL=0
MOVL C01843 V=800.0 PL=0
MOVL C01844 V=800.0 PL=0
MOVL C01845 V=800.0 PL=0
MOVL C01846 V=800.0 PL=0
MOVL C01847 V=800.0 PL=0
MOVL C01848 V=800.0 PL=0
MOVL C01849 V=800.0 PL=0
MOVL C01850 V=800.0 PL=0
MOVL C01851 V=800.0 PL=0
MOVL C01852 V=800.0 PL=0
MOVL C01853 V=800.0 PL=0
MOVL C01854 V=800.0 PL=0
MOVL C01855 V=800.0 PL=0
MOVL C01856 V=800.0 PL=0
MOVL C01857 V=800.0 PL=0
MOVL C01858 V=800.0 PL=0
MOVL C01859 V=800.0 PL=0
MOVL C01860 V=800.0 PL=0
MOVL C01861 V=800.0 PL=0
MOVL C01862 V=800.0 PL=0
MOVL C01863 V=800.0 PL=0
MOVL C01864 V=800.0 PL=0
MOVL C01865 V=800.0 PL=0
MOVL C01866 V=800.0 PL=0
MOVL C01867 V=800.0 PL=0
MOVL C01868 V=800.0 PL=0
MOVL C01869 V=800.0 PL=0
MOVL C01870 V=800.0 PL=0
MOVL C01871 V=800.0 PL=0
MOVL C01872 V=800.0 PL=0
MOVL C01873 V=800.0 PL=0
MOVL C01874 V=800.0 PL=0
MOVL C01875 V=800.0 PL=0
MOVL C01876 V=800.0 PL=0
MOVL C01877 V=800.0 PL=0
MOVL C01878 V=800.0 PL=0
MOVL C01879 V=800.0 PL=0
MOVL C01880 V=800.0 PL=0
MOVL C01881 V=800.0 PL=0
MOVL C01882 V=800.0 PL=0
MOVL C01883 V=800.0 PL=0
MOVL C01884 V=800.0 PL=0
MOVL C01885 V=800.0 PL=0
MOVL C01886 V=800.0 PL=0
MOVL C01887 V=800.0 PL=0
MOVL C01888 V=800.0 PL=0
MOVL C01889 V=800.0 PL=0
MOVL C01890 V=800.0 PL=0
MOVL C01891 V=800.0 PL=0
MOVL C01892 V=800.0 PL=0
MOVL C01893 V=800.0 PL=0
MOVL C01894 V=800.0 PL=0
MOVL C01895 V=800.0 PL=0
MOVL C01896 V=800.0 PL=0
MOVL C01897 V=800.0 PL=0
MOVL C01898 V=800.0 PL=0
MOVL C01899 V=800.0 PL=0
MOVL C01900 V=800.0 PL=0
MOVL C01901 V=800.0 PL=0
MOVL C01902 V=800.0 PL=0
MOVL C01903 V=800.0 PL=0
MOVL C01904 V=800.0 PL=0
MOVL C01905 V=800.0 PL=0
MOVL C01906 V=800.0 PL=0
MOVL C01907 V=800.0 PL=0
MOVL C01908 V=800.0 PL=0
MOVL C01909 V=800.0 PL=0
MOVL C01910 V=800.0 PL=0
MOVL C01911 V=800.0 PL=0
MOVL C01912 V=800.0 PL=0
MOVL C01913 V=800.0 PL=0
MOVL C01914 V=800.0 PL=0
MOVL C01915 V=800.0 PL=0
MOVL C01916 V=800.0 PL=0
MOVL C01917 V=800.0 PL=0
MOVL C01918 V=800.0 PL=0
MOVL C01919 V=800.0 PL=0
MOVL C01920 V=800.0 PL=0
MOVL C01921 V=800.0 PL=0
MOVL C01922 V=800.0 PL=0
MOVL C01923 V=800.0 PL=0
MOVL C01924 V=800.0 PL=0
MOVL C01925 V=800.0 PL=0
MOVL C01926 V=800.0 PL=0
MOVL C01927 V=800.0 PL=0
MOVL C01928 V=800.0 PL=0
MOVL C01929 V=800.0 PL=0
MOVL C01930 V=800.0 PL=0
MOVL C01931 V=800.0 PL=0
MOVL C01932 V=800.0 PL=0
MOVL C01933 V=800.0 PL=0
MOVL C01934 V=800.0 PL=0
MOVL C01935 V=800.0 PL=0
MOVL C01936 V=800.0 PL=0
MOVL C01937 V=800.0 PL=0
MOVL C01938 V=800.0 PL=0
MOVL C01939 V=800.0 PL=0
MOVL C01940 V=800.0 PL=0
MOVL C01941 V=800.0 PL=0
MOVL C01942 V=800.0 PL=0
MOVL C01943 V=800.0 PL=0
MOVL C01944 V=800.0 PL=0
MOVL C01945 V=800.0 PL=0
MOVL C01946 V=800.0 PL=0
MOVL C01947 V=800.0 PL=0
MOVL C01948 V=800.0 PL=0
MOVL C01949 V=800.0 PL=0
MOVL C01950 V=800.0 PL=0
MOVL C01951 V=800.0 PL=0
MOVL C01952 V=800.0 PL=0
MOVL C01953 V=800.0 PL=0
MOVL C01954 V=800.0 PL=0
MOVL C01955 V=800.0 PL=0
MOVL C01956 V=800.0 PL=0
MOVL C01957 V=800.0 PL=0
MOVL C01958 V=800.0 PL=0
MOVL C01959 V=800.0 PL=0
MOVL C01960 V=800.0 PL=0
MOVL C01961 V=800.0 PL=0
MOVL C01962 V=800.0 PL=0
MOVL C01963 V=800.0 PL=0
MOVL C01964 V=800.0 PL=0
MOVL C01965 V=800.0 PL=0
MOVL C01966 V=800.0 PL=0
MOVL C01967 V=800.0 PL=0
MOVL C01968 V=800.0 PL=0
MOVL C01969 V=800.0 PL=0
MOVL C01970 V=800.0 PL=0
MOVL C01971 V=800.0 PL=0
MOVL C01972 V=800.0 PL=0
MOVL C01973 V=800.0 PL=0
MOVL C01974 V=800.0 PL=0
MOVL C01975 V=800.0 PL=0
MOVL C01976 V=800.0 PL=0
MOVL C01977 V=800.0 PL=0
MOVL C01978 V=800.0 PL=0
MOVL C01979 V=800.0 PL=0
MOVL C01980 V=800.0 PL=0
MOVL C01981 V=800.0 PL=0
MOVL C01982 V=800.0 PL=0
MOVL C01983 V=800.0 PL=0
MOVL C01984 V=800.0 PL=0
MOVL C01985 V=800.0 PL=0
MOVL C01986 V=800.0 PL=0
MOVL C01987 V=800.0 PL=0
MOVL C01988 V=800.0 PL=0
MOVL C01989 V=800.0 PL=0
MOVL C01990 V=800.0 PL=0
MOVL C01991 V=800.0 PL=0
MOVL C01992 V=800.0 PL=0
MOVL C01993 V=800.0 PL=0
MOVL C01994 V=800.0 PL=0
MOVL C01995 V=800.0 PL=0
MOVL C01996 V=800.0 PL=0
MOVL C01997 V=800.0 PL=0
MOVL C01998 V=800.0 PL=0
MOVL C01999 V=800.0 PL=0
MOVL C02000 V=800.0 PL=0
MOVL C02001 V=800.0 PL=0
MOVL C02002 V=800.0 PL=0
MOVL C02003 V=800.0 PL=0
MOVL C02004 V=800.0 PL=0
MOVL C02005 V=800.0 PL=0
MOVL C02006 V=800.0 PL=0
MOVL C02007 V=800.0 PL=0
MOVL C02008 V=800.0 PL=0
MOVL C02009 V=800.0 PL=0
MOVL C02010 V=800.0 PL=0
MOVL C02011 V=800.0 PL=0
MOVL C02012 V=800.0 PL=0
MOVL C02013 V=800.0 PL=0
MOVL C02014 V=800.0 PL=0
MOVL C02015 V=800.0 PL=0
MOVL C02016 V=800.0 PL=0
MOVL C02017 V=800.0 PL=0
MOVL C02018 V=800.0 PL=0
MOVL C02019 V=800.0 PL=0
MOVL C02020 V=800.0 PL=0
MOVL C02021 V=800.0 PL=0
MOVL C02022 V=800.0 PL=0
MOVL C02023 V=800.0 PL=0
MOVL C02024 V=800.0 PL=0
MOVL C02025 V=800.0 PL=0
MOVL C02026 V=800.0 PL=0
MOVL C02027 V=800.0 PL=0
MOVL C02028 V=800.0 PL=0
MOVL C02029 V=800.0 PL=0
MOVL C02030 V=800.0 PL=0
MOVL C02031 V=800.0 PL=0
MOVL C02032 V=800.0 PL=0
MOVL C02033 V=800.0 PL=0
MOVL C02034 V=800.0 PL=0
MOVL C02035 V=800.0 PL=0
MOVL C02036 V=800.0 PL=0
MOVL C02037 V=800.0 PL=0
MOVL C02038 V=800.0 PL=0
MOVL C02039 V=800.0 PL=0
MOVL C02040 V=800.0 PL=0
MOVL C02041 V=800.0 PL=0
MOVL C02042 V=800.0 PL=0
MOVL C02043 V=800.0 PL=0
MOVL C02044 V=800.0 PL=0
MOVL C02045 V=800.0 PL=0
MOVL C02046 V=800.0 PL=0
MOVL C02047 V=800.0 PL=0
MOVL C02048 V=800.0 PL=0
MOVL C02049 V=800.0 PL=0
MOVL C02050 V=800.0 PL=0
MOVL C02051 V=800.0 PL=0
MOVL C02052 V=800.0 PL=0
MOVL C02053 V=800.0 PL=0
MOVL C02054 V=800.0 PL=0
MOVL C02055 V=800.0 PL=0
MOVL C02056 V=800.0 PL=0
MOVL C02057 V=800.0 PL=0
MOVL C02058 V=800.0 PL=0
MOVL C02059 V=800.0 PL=0
MOVL C02060 V=800.0 PL=0
MOVL C02061 V=800.0 PL=0
MOVL C02062 V=800.0 PL=0
MOVL C02063 V=800.0 PL=0
MOVL C02064 V=800.0 PL=0
MOVL C02065 V=800.0 PL=0
MOVL C02066 V=800.0 PL=0
MOVL C02067 V=800.0 PL=0
MOVL C02068 V=800.0 PL=0
MOVL C02069 V=800.0 PL=0
MOVL C02070 V=800.0 PL=0
MOVL C02071 V=800.0 PL=0
MOVL C02072 V=800.0 PL=0
MOVL C02073 V=800.0 PL=0
MOVL C02074 V=800.0 PL=0
MOVL C02075 V=800.0 PL=0
MOVL C02076 V=800.0 PL=0
MOVL C02077 V=800.0 PL=0
MOVL C02078 V=800.0 PL=0
MOVL C02079 V=800.0 PL=0
MOVL C02080 V=800.0 PL=0
MOVL C02081 V=800.0 PL=0
MOVL C02082 V=800.0 PL=0
MOVL C02083 V=800.0 PL=0
MOVL C02084 V=800.0 PL=0
MOVL C02085 V=800.0 PL=0
MOVL C02086 V=800.0 PL=0
MOVL C02087 V=800.0 PL=0
MOVL C02088 V=800.0 PL=0
MOVL C02089 V=800.0 PL=0
MOVL C02090 V=800.0 PL=0
MOVL C02091 V=800.0 PL=0
MOVL C02092 V=800.0 PL=0
MOVL C02093 V=800.0 PL=0
MOVL C02094 V=800.0 PL=0
MOVL C02095 V=800.0 PL=0
MOVL C02096 V=800.0 PL=0
MOVL C02097 V=800.0 PL=0
MOVL C02098 V=800.0 PL=0
MOVL C02099 V=800.0 PL=0
MOVL C02100 V=800.0 PL=0
MOVL C02101 V=800.0 PL=0
MOVL C02102 V=800.0 PL=0
MOVL C02103 V=800.0 PL=0
MOVL C02104 V=800.0 PL=0
MOVL C02105 V=800.0 PL=0
MOVL C02106 V=800.0 PL=0
MOVL C02107 V=800.0 PL=0
MOVL C02108 V=800.0 PL=0
MOVL C02109 V=800.0 PL=0
MOVL C02110 V=800.0 PL=0
MOVL C02111 V=800.0 PL=0
MOVL C02112 V=800.0 PL=0
MOVL C02113 V=800.0 PL=0
MOVL C02114 V=800.0 PL=0
MOVL C02115 V=800.0 PL=0
MOVL C02116 V=800.0 PL=0
MOVL C02117 V=800.0 PL=0
MOVL C02118 V=800.0 PL=0
MOVL C02119 V=800.0 PL=0
MOVL C02120 V=800.0 PL=0
MOVL C02121 V=800.0 PL=0
MOVL C02122 V=800.0 PL=0
MOVL C02123 V=800.0 PL=0
MOVL C02124 V=800.0 PL=0
MOVL C02125 V=800.0 PL=0
MOVL C02126 V=800.0 PL=0
MOVL C02127 V=800.0 PL=0
MOVL C02128 V=800.0 PL=0
MOVL C02129 V=800.0 PL=0
